// TIA Portal project "Bachelor _Project" (V17)
// By Soroush Tehranchi

(* hardware
DEVICE "S7-300/ET200M station_1"  S7-300 station
   slot 0: "Rail_0"  Rail  6ES7 390-1***0-0AA0
   slot 1: "PS 307 5A Outdoor_1"  PS 307 5A Outdoor  6ES7 307-1EA80-0AA0
   slot 1: "Rail_1"  Rail  6ES7 390-1***0-0AA0
   slot 1: "PS 307 5A_1"  PS 307 5A  6ES7 307-1EA01-0AA0
   slot 2: "PLC Siemens S7-300"  CPU 317-2 PN/DP  6ES7 317-2EK14-0AB0  V3.2
      slot 2: "PROFINET interface_1"  PN-IO
         slot 1: "Port_1"  Port
         slot 2: "Port_2"  Port
   slot 3: "IM 365_1"  IM 365  6ES7 365-0BA01-0AA0
      slot 1: "IM send/receive interface_1"  6ES7 365-0BA00-0AA0
   slot 3: "IM 365_1"  IM 365  6ES7 365-0BA01-0AA0
      slot 1: "IM send/receive interface_1"  6ES7 365-0BA00-0AA0
   slot 4: "DI 16x24VDC_1"  DI16 x 24VDC  6ES7 321-1BH02-0AA0
   slot 4: "DO 16x24VDC/0.5A_1"  DO16 x 24VDC / 0.5A  6ES7 322-1BH01-0AA0
   slot 5: "DI 16x24VDC_2"  DI16 x 24VDC  6ES7 321-1BH02-0AA0
   slot 5: "DO 16x24VDC/0.5A_2"  DO16 x 24VDC / 0.5A  6ES7 322-1BH01-0AA0
   slot 6: "DI 16x24VDC_3"  DI16 x 24VDC  6ES7 321-1BH02-0AA0
   slot 6: "DO 16x24VDC/0.5A_3"  DO16 x 24VDC / 0.5A  6ES7 322-1BH01-0AA0
   slot 7: "DI 16x24VDC_4"  DI16 x 24VDC  6ES7 321-1BH02-0AA0
   slot 7: "DO 16x24VDC/0.5A_4"  DO16 x 24VDC / 0.5A  6ES7 322-1BH01-0AA0
   slot 8: "AI 8x12BIT_1"  AI8 x 12 bits  6ES7 331-7KF02-0AB0
   slot 8: "FM 350-1 Counter_1"  FM 350-1 Counter  6ES7 350-1AH03-0AE0
   slot 9: "AI 8x12BIT_2"  AI8 x 12 bits  6ES7 331-7KF02-0AB0
   slot 9: "AI 8x12BIT_1"  AI8 x 12 bits  6ES7 331-7KF02-0AB0
   slot 10: "AI 8x12BIT_3"  AI8 x 12 bits  6ES7 331-7KF02-0AB0
   slot 10: "AI 8x12BIT_2"  AI8 x 12 bits  6ES7 331-7KF02-0AB0
   slot 11: "AO 8x12BIT_1"  AO8 x 12 bits  6ES7 332-5HF00-0AB0
   slot 11: "AO 8x12BIT_1"  AO8 x 12 bits  6ES7 332-5HF00-0AB0
DEVICE "HMI_1"  TP1200 Comfort
   slot 0: "HMI_1"  TP1200 Comfort  6AV2 124-0MC01-0AX0  17.0.0.0
   slot 1: "HMI_RT_1"  TP1200 Comfort  6AV2 124-0MC01-0AX0  17.0.0.0
   slot 5: "HMI_1.IE_CP_1"  PROFINET Interface  17.0.0.0
      slot 1: "PROFINET Interface_1"  PROFINET Interface
         slot 1: "Port_1"  Port
         slot 2: "Port_2"  Port
   slot 7: "HMI_1.MPI/DP_CP_1"  MPI/DP Interface  17.0.0.0
*)

// ===== PLC "PLC Siemens S7-300"  CPU 317-2 PN/DP =====

VAR_GLOBAL   // PLC tag table "Default tag table"
   "blue assembler convoyer timer" AT %T0 : Timer;
   "Machinings 2 timer(1)" AT %T1 : Timer;
   "Machinings 2 timer" AT %T2 : Timer;
   "Machinings 3 timer" AT %T3 : Timer;
   "Machinings 4 timer" AT %T4 : Timer;
   "station 1 counter" AT %C0 : Counter;
   "count sort line" AT %C1 : Counter;
   "count up sort" AT %M1.4 : Bool;
   "in position sort" AT %M1.5 : Bool;
   "Green base memory" AT %M1.6 : Bool;
   "sort convoyer edje" AT %M1.7 : Bool;
   "Green base counter" AT %C2 : Counter;
   "Blue base counter" AT %C3 : Counter;
   "Green lid counter" AT %C4 : Counter;
   "Blue lid counter" AT %C5 : Counter;
   "Green base counter number" AT %MW100 : Int;
   "Blue base counter number" AT %MW102 : Int;
   "Green lid counter number" AT %MW104 : Int;
   "Blue lid counter number" AT %MW106 : Int;
   "pusher edje 6" AT %M2.0 : Bool;
   "pusher edje 5" AT %M2.1 : Bool;
   "pusher edje 3" AT %M2.2 : Bool;
   "pusher edje 2" AT %M2.3 : Bool;
   "sort line counter number" AT %MW108 : Int;
   "encoder edje5" AT %M3.2 : Bool;
   "encoder edje6" AT %M3.3 : Bool;
   "encoder edje7" AT %M3.4 : Bool;
   "encoder edje8" AT %M3.5 : Bool;
   "encoder edje9" AT %M3.6 : Bool;
   "encoder edje10" AT %M3.7 : Bool;
   "encoder edje11" AT %M4.0 : Bool;
   "encoder edje12" AT %M4.1 : Bool;
   "encoder edje13" AT %M4.2 : Bool;
   "encoder edje14" AT %M4.3 : Bool;
   "encoder edje15" AT %M4.4 : Bool;
   "encoder edje16" AT %M4.5 : Bool;
   "Blue lid memory" AT %M4.6 : Bool;
   "green lid memory" AT %M4.7 : Bool;
   "initial assembler 2" AT %M6.7 : Bool;
   "initial assembler 1" AT %M6.6 : Bool;
   "Packaging Green  Clamp Sensor" AT %I3.6 : Bool;
   "green assembler convoyer timer" AT %T5 : Timer;
   "packing 1 uptimer" AT %T6 : Timer;
   "counter packing 1 uptime" AT %C6 : Counter;
   "Packing blue uptime" AT %T7 : Timer;
   "uptime blue packing" AT %C7 : Counter;
   "Item in blue pack" AT %C8 : Counter;
   "Item in green pack" AT %C9 : Counter;
   "Blue pack produced" AT %C10 : Counter;
   "green pack produced" AT %C11 : Counter;
   "blue product" AT %C12 : Counter;
   "green product" AT %C13 : Counter;
   "Assembler uptime blue" AT %T8 : Timer;
   "Blue Assembler uptime" AT %C14 : Counter;
   "green assembler uptimer" AT %T9 : Timer;
   "green assembler uptime" AT %C15 : Counter;
   "main convoyer uptimer" AT %T10 : Timer;
   "main convoyer uptime" AT %C16 : Counter;
   "crane uptimer" AT %T12 : Timer;
   "crane uptime" AT %C17 : Counter;
END_VAR

VAR_GLOBAL   // PLC tag table "Inputs"
   "Base  Blue Positioner (Clamped)" AT %I0.0 : Bool;
   "Base  Blue Positioner (Limit)" AT %I0.1 : Bool;
   "Base  Green Positioner (Clamped)" AT %I0.2 : Bool;
   "Base  Green Positioner (Limit)" AT %I0.3 : Bool;
   "Base Blue Clamp Sensor" AT %I0.4 : Bool;
   "Base Green Clamp Sensor" AT %I0.5 : Bool;
   "Blue Pusher Base  (Front Limit)" AT %I0.6 : Bool;
   "Blue Pusher Base (Back Limit)" AT %I0.7 : Bool;
   "Blue Pusher Lid (Back Limit)" AT %I1.0 : Bool;
   "Blue Pusher Lid (Front Limit)" AT %I1.1 : Bool;
   "Green Pusher Base  (Front Limit)" AT %I1.2 : Bool;
   "Green Pusher Base (Back Limit)" AT %I1.3 : Bool;
   "Green Pusher Lid (Back Limit)" AT %I1.4 : Bool;
   "Green Pusher Lid (Front Limit)" AT %I1.5 : Bool;
   "Lid  Blue Positioner (Clamped)" AT %I1.6 : Bool;
   "Lid  Green Positioner (Clamped)" AT %I1.7 : Bool;
   "Lid Blue Clamp Sensor" AT %I2.0 : Bool;
   "Lid Green Clamp Sensor" AT %I2.1 : Bool;
   "Machining Center 1 (Opened)" AT %I2.2 : Bool;
   "Machining Center 2 (Opened)" AT %I2.3 : Bool;
   "Machining Center 3 (Opened)" AT %I2.4 : Bool;
   "Machining Center 4 (Opened)" AT %I2.5 : Bool;
   "Machining Center 1 (Is Busy)" AT %I2.6 : Bool;
   "Machining Center 2 (Is Busy)" AT %I2.7 : Bool;
   "Machining Center 3 (Is Busy)" AT %I3.0 : Bool;
   "Machining Center 4 (Is Busy)" AT %I3.1 : Bool;
   "Packaging Blue (Limit)" AT %I3.2 : Bool;
   "Packaging Blue Palet Sensor" AT %I3.3 : Bool;
   "Packaging Blue(Clamped)" AT %I3.4 : Bool;
   "Packaging Green  (Limit)" AT %I3.5 : Bool;
   "Packaging Blue Clamp Sensor" AT %I3.7 : Bool;
   "Packaging Green  Palet Sensor" AT %I4.0 : Bool;
   "Packaging Green (Clamped)" AT %I4.1 : Bool;
   "Pick & Place 1 (C Limit) packaging" AT %I4.2 : Bool;
   "Pick & Place 2 (C Limit) packaging" AT %I4.3 : Bool;
   "Assmebler 1  grabed" AT %I4.4 : Bool;
   "Assmebler 2  grabed" AT %I4.5 : Bool;
   "Pick & Place 1 (Box Detected) packaging" AT %I5.4 : Bool;
   "Pick & Place 2 (Box Detected) packaging" AT %I5.5 : Bool;
   "Stacker Crane 1 Moving-X" AT %I6.2 : Bool;
   "Stacker Crane 1 Moving-Z" AT %I6.3 : Bool;
   "Stacker Crane 1 Left Limit" AT %I6.4 : Bool;
   "Stacker Crane 1 Right Limit" AT %I6.5 : Bool;
   "Stacker Crane 1 Middle Limit" AT %I6.6 : Bool;
   "Turntable 1 (Limit 0)" AT %I6.7 : Bool;
   "Turntable 1 (Limit 90)" AT %I7.0 : Bool;
   "Turntable 1 (Back Limit)" AT %I7.1 : Bool;
   "Turntable 1 (Front Limit)" AT %I7.2 : Bool;
   "Sort Convoyer Encoder Signal A" AT %I8.0 : Bool;
   "Sort Convoyer Encoder Signal B" AT %I8.1 : Bool;
   "Assemble Base Blue Convoyer" AT %Q0.1 : Bool;
   "Assemble Base Green Convoyer" AT %Q0.2 : Bool;
   "Assemble Lid Blue Convoyer" AT %Q0.3 : Bool;
   "Assemble Lid Green Convoyer" AT %Q0.4 : Bool;
   "Base  Blue Positioner  (Raise)" AT %Q0.5 : Bool;
   "Base  Blue Positioner (Clamp)" AT %Q0.6 : Bool;
   "Base  Green Positioner (Clamp)" AT %Q0.7 : Bool;
   "Base  Green Positioner (Raise)" AT %Q1.0 : Bool;
   "Blue Assemble Exit Convoyer 1" AT %Q1.1 : Bool;
   "Blue Assemble Exit Convoyer 2" AT %Q1.2 : Bool;
   "Blue Pusher Base" AT %Q1.3 : Bool;
   "Blue Pusher Lid" AT %Q1.4 : Bool;
   "Exit Convoyer" AT %Q1.5 : Bool;
   "Green Assemble Exit Convoyer" AT %Q1.6 : Bool;
   "Green Pusher Base" AT %Q1.7 : Bool;
   "Green Pusher Lid" AT %Q2.0 : Bool;
   "Lid  Blue Positioner (Clamp)" AT %Q2.2 : Bool;
   "Lid  Green Positioner (Clamp)" AT %Q2.3 : Bool;
   "Machining1 Exit Convoyer" AT %Q2.5 : Bool;
   "Machining2 Exit Convoyer" AT %Q2.6 : Bool;
   "Machining3 Exit Convoyer" AT %Q2.7 : Bool;
   "Machining4 Exit Convoyer" AT %Q3.0 : Bool;
   "Machining1 Entry Convoyer" AT %Q3.1 : Bool;
   "Machining2 Entry Convoyer" AT %Q3.2 : Bool;
   "Machining3 Entry Convoyer" AT %Q3.3 : Bool;
   "Machining4 Entry Convoyer" AT %Q3.4 : Bool;
   "Machinings Exit Convoyer 1" AT %Q3.5 : Bool;
   "Machinings Exit Convoyer 2" AT %Q3.6 : Bool;
   "Machinings Exit Convoyer 3" AT %Q3.7 : Bool;
   "Packaging Blue (Raise)" AT %Q4.0 : Bool;
   "Packaging Blue Convoyer" AT %Q4.1 : Bool;
   "Packaging Blue Exit Convoyer 1" AT %Q4.2 : Bool;
   "Packaging Blue Exit Convoyer 2" AT %Q4.3 : Bool;
   "Packaging Blue Exit Convoyer 3" AT %Q4.4 : Bool;
   "Packaging Blue(Clamp)" AT %Q4.5 : Bool;
   "Packaging Green (Clamp)" AT %Q4.6 : Bool;
   "Packaging Green (Raise)" AT %Q4.7 : Bool;
   "Packaging Green Convoyer" AT %Q5.0 : Bool;
   "Packaging Green Exit Convoyer" AT %Q5.1 : Bool;
   "Two-Axis Pick & Place 1 (Grab)" AT %Q5.2 : Bool;
   "Two-Axis Pick & Place 2 (Grab)" AT %Q5.3 : Bool;
   "Two-Axis Pick & Place 1 Rotate CW" AT %Q5.4 : Bool;
   "Pick & Place 1 C(+) packaging" AT %Q5.5 : Bool;
   "Pick & Place 2 C(+) packaging" AT %Q5.6 : Bool;
   "Pick & Place 1 (Grab) packaging" AT %Q5.7 : Bool;
   "Two-Axis Pick & Place 2 Rotate CW" AT %Q6.0 : Bool;
   "Two-Axis Pick & Place 1 Gripper CW" AT %Q6.1 : Bool;
   "Two-Axis Pick & Place 2 Gripper CW" AT %Q6.2 : Bool;
   "Pick & Place 2 (Grab) packaging" AT %Q6.6 : Bool;
   "Sort Convoyer" AT %Q6.7 : Bool;
   "Stacker Crane 1 Lift" AT %Q7.0 : Bool;
   "Stacker Crane 1 (Left)" AT %Q7.1 : Bool;
   "Stacker Crane 1 (Right)" AT %Q7.2 : Bool;
   "Turntable 1 Turn" AT %Q7.4 : Bool;
   "Turntable 1 Roll (+)" AT %Q7.5 : Bool;
   "Turntable 1 Roll (-)" AT %Q7.6 : Bool;
   "Vision Sensor 1 (Value)" AT %ID100 : DInt;
   "Pick & Place 2 Z Position (V) packaging" AT %ID104 : Real;
   "Pick & Place 2 Y Position (V) packaging" AT %ID108 : Real;
   "Pick & Place 2 X Position (V) packaging" AT %ID112 : Real;
   "Pick & Place 1 Z Position (V) packaging" AT %ID116 : Real;
   "Pick & Place 1 Y Position (V) packaging" AT %ID120 : Real;
   "Pick & Place 1 X Position (V) packaging" AT %ID124 : Real;
   "Machining Center 4 (Progress)" AT %ID128 : DInt;
   "Machining Center 3 (Progress)" AT %ID132 : DInt;
   "Machining Center 2 (Progress)" AT %ID136 : DInt;
   "Machining Center 1 (Progress)" AT %ID140 : DInt;
   "Vision Sensor 2 (Value)" AT %ID144 : DInt;
   "Vision Sensor 3 (Value)" AT %ID148 : DInt;
   "Vision Sensor 4 (Value)" AT %ID152 : DInt;
   "Two-Axis Pick & Place 1 X Position (V)" AT %ID156 : Real;
   "Two-Axis Pick & Place 1 Z Position (V)" AT %ID160 : Real;
   "Two-Axis Pick & Place 2 X Position (V)" AT %ID164 : Real;
   "Two-Axis Pick & Place 2 Z Position (V)" AT %ID168 : Real;
   "Pick & Place 1 Y Set Point(V) packaging" AT %QD100 : Real;
   "Pick & Place 2 Y Set Point(V) packaging" AT %QD104 : Real;
   "Pick & Place 1 X Set Point (V) packaging" AT %QD108 : Real;
   "Pick & Place 1 Z Set Point (V) packaging" AT %QD112 : Real;
   "Pick & Place 2 X Set Point (V) packaging" AT %QD116 : Real;
   "Pick & Place 2 Z Set Point (V) packaging" AT %QD120 : Real;
   "Stacker Crane 1 Target Position" AT %QD124 : DInt;
   "Two-Axis Pick & Place 1 X Set Point (V)" AT %QD128 : Real;
   "Two-Axis Pick & Place 1 Z Set Point (V)" AT %QD132 : Real;
   "Two-Axis Pick & Place 2 X Set Point (V)" AT %QD136 : Real;
   "Two-Axis Pick & Place 2 Z Set Point (V)" AT %QD140 : Real;
   "two axis  1 assembler rotating" AT %I4.6 : Bool;
   "two axis  2 assembler rotating" AT %I4.7 : Bool;
   "Capacitive Sensor Exit line 1" AT %I5.0 : Bool;
   "Capacitive Sensor Exit line 2" AT %I5.1 : Bool;
   "cran capacetive sensor" AT %I5.2 : Bool;
   "packaging to turn table convoyer" AT %Q2.1 : Bool;
   "Loading convoyer -" AT %Q0.0 : Bool;
   "Loading convoyer +" AT %Q2.4 : Bool;
   "Emitter 6" AT %Q6.3 : Bool;
   "Emmiter5" AT %Q6.4 : Bool;
END_VAR

VAR_GLOBAL   // PLC tag table "memory"
   "start_mach_entry_conv" AT %M0.0 : Bool;   // start machine center convoyer
   "reset convoyers" AT %M0.1 : Bool;
   "Machining Center busy1" AT %M0.2 : Bool;
   "Machining Center busy2" AT %M0.3 : Bool;
   "Machining Center busy3" AT %M0.4 : Bool;
   "Machining Center busy4" AT %M0.5 : Bool;
   "Machining Center busy1 convoyer" AT %M0.6 : Bool;
   "Machining Center busy2 convoyer" AT %M0.7 : Bool;
   "Machining Center busy3 convoyer" AT %M1.0 : Bool;
   "Machining Center busy4 convoyer" AT %M1.1 : Bool;
   "count down memory" AT %M1.2 : Bool;
   "count up memory" AT %M1.3 : Bool;
   "reset sorter" AT %M3.1 : Bool;
   "blue lid clamp sensor edje" AT %M5.0 : Bool;
   "blue base clamp sensor edje" AT %M5.1 : Bool;
   "green lid clamp sensor edje" AT %M5.2 : Bool;
   "green base clamp sensor edje" AT %M5.3 : Bool;
   "line 1 ready" AT %M5.4 : Bool;
   "line 2 ready" AT %M5.5 : Bool;
   "line 3 ready" AT %M5.6 : Bool;
   "line 4 ready" AT %M5.7 : Bool;
   "assemble 1 complet" AT %M6.0 : Bool;
   "assemble 2 complet" AT %M6.1 : Bool;
   "reset convoyers assembler" AT %M6.2 : Bool;
   "ready 1 edje" AT %M6.3 : Bool;
   "blue lid clamp sensor edje2" AT %M6.4 : Bool;
   "blue base positioner rise adje up" AT %M6.5 : Bool;
   "blue base positioner rise adje down" AT %M7.0 : Bool;
   "blue base clamp sensor edje2" AT %M7.1 : Bool;
   "green lid clamp sensor edje2" AT %M7.2 : Bool;
   "green  base positioner rise adje up" AT %M7.3 : Bool;
   "green base positioner rise adje down" AT %M7.4 : Bool;
   "green  base clamp sensor edje2" AT %M7.5 : Bool;
   "Packaging Green  Clamp Sensor edje" AT %M7.6 : Bool;
   "Packaging Green  Clamp Senso edje" AT %M7.7 : Bool;
   "packing 1 done" AT %M8.0 : Bool;
   "packing 2 done" AT %M8.1 : Bool;
   "Packaging Blue Palet Sensor edje" AT %M8.2 : Bool;
   "exit convoyer packing blue ready" AT %M8.3 : Bool;
   "entry convoyer packing blue ready" AT %M8.4 : Bool;
   "Packaging Blue Palet Sensor edje2" AT %M8.5 : Bool;
   "Packaging Green  Clamp Sensor edje 2" AT %M8.6 : Bool;
   "ready to pack 1" AT %M8.7 : Bool;
   "ready to pack 2" AT %M9.0 : Bool;
   "reset packer 1" AT %M9.1 : Bool;
   "reset packer 2" AT %M9.2 : Bool;
   "Capacitive Sensor Exit line 1 edje" AT %M9.3 : Bool;
   "Capacitive Sensor Exit line 2 edje" AT %M9.4 : Bool;
   "Packaging Blue Clamp Sensor edje 2" AT %M9.5 : Bool;
   "entry convoyer packing green ready" AT %M9.6 : Bool;
   "Packaging green Palet Sensor edje" AT %M9.7 : Bool;
   "exit convoyer packing green ready" AT %M10.0 : Bool;
   "Packaging green Palet Sensor edje2" AT %M10.1 : Bool;
   "Load to storage" AT %M10.2 : Bool;
   "Capacitive Sensor Exit line 2 edje(1)" AT %M10.3 : Bool;
   "deploy" AT %M10.4 : Bool;
   "user target position" AT %MD20 : DInt;
   "product type" AT %MW24 : Int;   // 0 empty 1green 2 blue
   "blue item stored" AT %MW26 : Int;
   "green item stored" AT %MW28 : Int;
   "cap" AT %MW30 : Int;
END_VAR

// folder: Packaging

DATA_BLOCK "Packaging system_DB"   // DB3
{ S7_Optimized_Access := 'FALSE' }
VERSION : 0.1
// stored: InstanceOfName Packaging systemBlue
"Packaging systemBlue"
BEGIN
END_DATA_BLOCK

DATA_BLOCK "Packaging system2_DB"   // DB4
{ S7_Optimized_Access := 'FALSE' }
VERSION : 0.1
// stored: InstanceOfName Packaging system Green
"Packaging system Green"
BEGIN
END_DATA_BLOCK

// folder: Sort And Assemble

DATA_BLOCK "Assembler_devic_DB"   // DB1
{ S7_Optimized_Access := 'FALSE' }
VERSION : 0.1
// stored: InstanceOfName Assembler_devic
"Assembler_devic"
BEGIN
END_DATA_BLOCK

DATA_BLOCK "Assembler_devic_DB_1"   // DB2
{ S7_Optimized_Access := 'FALSE' }
VERSION : 0.1
// stored: InstanceOfName Assembler_devic
"Assembler_devic"
BEGIN
END_DATA_BLOCK

// folder: Storage System

DATA_BLOCK "Turntable_DB"   // DB5
{ S7_Optimized_Access := 'FALSE' }
VERSION : 0.1
// stored: InstanceOfName Turntable
"Turntable"
BEGIN
END_DATA_BLOCK

DATA_BLOCK "Storage"   // DB6
{ S7_Optimized_Access := 'FALSE' }
VERSION : 0.1
   VAR
      status : Array[0..53] of Bool;
      cap : Int;
      "product type" : Array[0..53] of Int;
   END_VAR
BEGIN
   "product type"[1] := 0;
   "product type"[2] := 0;
END_DATA_BLOCK

DATA_BLOCK "stacker_DB"   // DB7
{ S7_Optimized_Access := 'FALSE' }
VERSION : 0.1
// stored: InstanceOfName stacker
"stacker"
BEGIN
END_DATA_BLOCK

// folder: (top level)

ORGANIZATION_BLOCK "Main"   // OB1, LAD
TITLE = "Main Program Sweep (Cycle)"
{ S7_Optimized_Access := 'FALSE' }
VERSION : 0.1
   VAR_TEMP
      OB1_EV_CLASS : Byte;   // Bits 0-3 = 1 (Coming event), Bits 4-7 = 1 (Event class 1)
      OB1_SCAN_1 : Byte;   // 1 (Cold restart scan 1 of OB 1), 3 (Scan 2-n of OB 1)
      OB1_PRIORITY : Byte;   // Priority of OB Execution
      OB1_OB_NUMBR : Byte;   // 1 (Organization block 1, OB1)
      OB1_RESERVED_1 : Byte;   // Reserved for system
      OB1_RESERVED_2 : Byte;   // Reserved for system
      OB1_PREV_CYCLE : Int;   // Cycle time of previous OB1 scan (milliseconds)
      OB1_MIN_CYCLE : Int;   // Minimum cycle time of OB1 (milliseconds)
      OB1_MAX_CYCLE : Int;   // Maximum cycle time of OB1 (milliseconds)
      OB1_DATE_TIME : Date_And_Time;   // Date and time OB1 started
   END_VAR
BEGIN

REGION Network 1: Machining Center
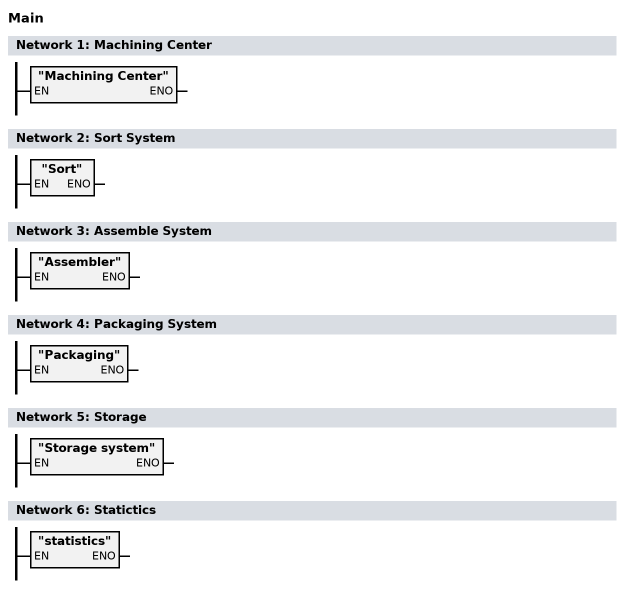
   RUNG wire#powerrail
      "Machining Center"()
   END_RUNG
   // the same network as SCL:
   "Machining Center"();
END_REGION

REGION Network 2: Sort System
   RUNG wire#powerrail
      "Sort"()
   END_RUNG
   // the same network as SCL:
   "Sort"();
END_REGION

REGION Network 3: Assemble System
   RUNG wire#powerrail
      "Assembler"()
   END_RUNG
   // the same network as SCL:
   "Assembler"();
END_REGION

REGION Network 4: Packaging System
   RUNG wire#powerrail
      "Packaging"()
   END_RUNG
   // the same network as SCL:
   "Packaging"();
END_REGION

REGION Network 5: Storage
   RUNG wire#powerrail
      "Storage system"()
   END_RUNG
   // the same network as SCL:
   "Storage system"();
END_REGION

REGION Network 6: Statictics
   RUNG wire#powerrail
      "statistics"()
   END_RUNG
   // the same network as SCL:
   "statistics"();
END_REGION
END_ORGANIZATION_BLOCK

// folder: Machining Center

FUNCTION "Machining Center" : Void   // FC1, LAD
TITLE = Machining Center
{ S7_Optimized_Access := 'FALSE' }
VERSION : 0.1
// This FC manage Entry Convoyer and exit convoyer
BEGIN

REGION Network 1: Entry Convoyers
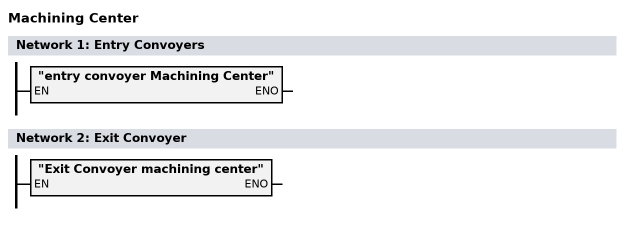
   RUNG wire#powerrail
      "entry convoyer Machining Center"()
   END_RUNG
   // the same network as SCL:
   "entry convoyer Machining Center"();
END_REGION

REGION Network 2: Exit Convoyer
   RUNG wire#powerrail
      "Exit Convoyer machining center"()
   END_RUNG
   // the same network as SCL:
   "Exit Convoyer machining center"();
END_REGION
END_FUNCTION

FUNCTION "entry convoyer Machining Center" : Void   // FC2, LAD
{ S7_Optimized_Access := 'FALSE' }
VERSION : 0.1
BEGIN

REGION Network 1
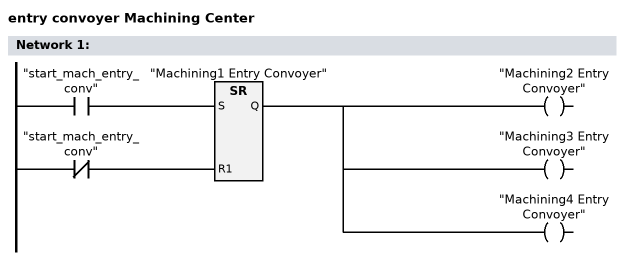
   RUNG wire#powerrail
      Contact( "start_mach_entry_conv" )
      S_SR(operand := "Machining1 Entry Convoyer", r1 := wire#w1)
      wire#w2
      Coil( "Machining2 Entry Convoyer" )
   END_RUNG
   RUNG wire#powerrail
      I_Contact( "start_mach_entry_conv" )
   END_RUNG wire#w1
   RUNG wire#w2
      Coil( "Machining3 Entry Convoyer" )
   END_RUNG
   RUNG wire#w2
      Coil( "Machining4 Entry Convoyer" )
   END_RUNG
   // the same network as SCL:
   IF "start_mach_entry_conv" THEN
       "Machining1 Entry Convoyer" := TRUE;   // SR flip-flop
   END_IF;
   IF NOT "start_mach_entry_conv" THEN "Machining1 Entry Convoyer" := FALSE; END_IF;
   "Machining2 Entry Convoyer" := "Machining1 Entry Convoyer";
   "Machining3 Entry Convoyer" := "Machining1 Entry Convoyer";
   "Machining4 Entry Convoyer" := "Machining1 Entry Convoyer";
END_REGION
END_FUNCTION

FUNCTION "Exit Convoyer machining center" : Void   // FC3, LAD
{ S7_Optimized_Access := 'FALSE' }
VERSION : 0.1
   VAR_TEMP   // added for the SCL form of the ladder/FBD networks
      _w1 : Bool;
      _w2 : Bool;
      _w3 : Bool;
      _w4 : Bool;
      _w5 : Bool;
      _w6 : Bool;
      _w7 : Bool;
      _w8 : Bool;
      _w9 : Bool;
      _w10 : Bool;
      _w11 : Bool;
      _s5time1 : S5Time;
   END_VAR
BEGIN

REGION Network 1: Exit Convoyers
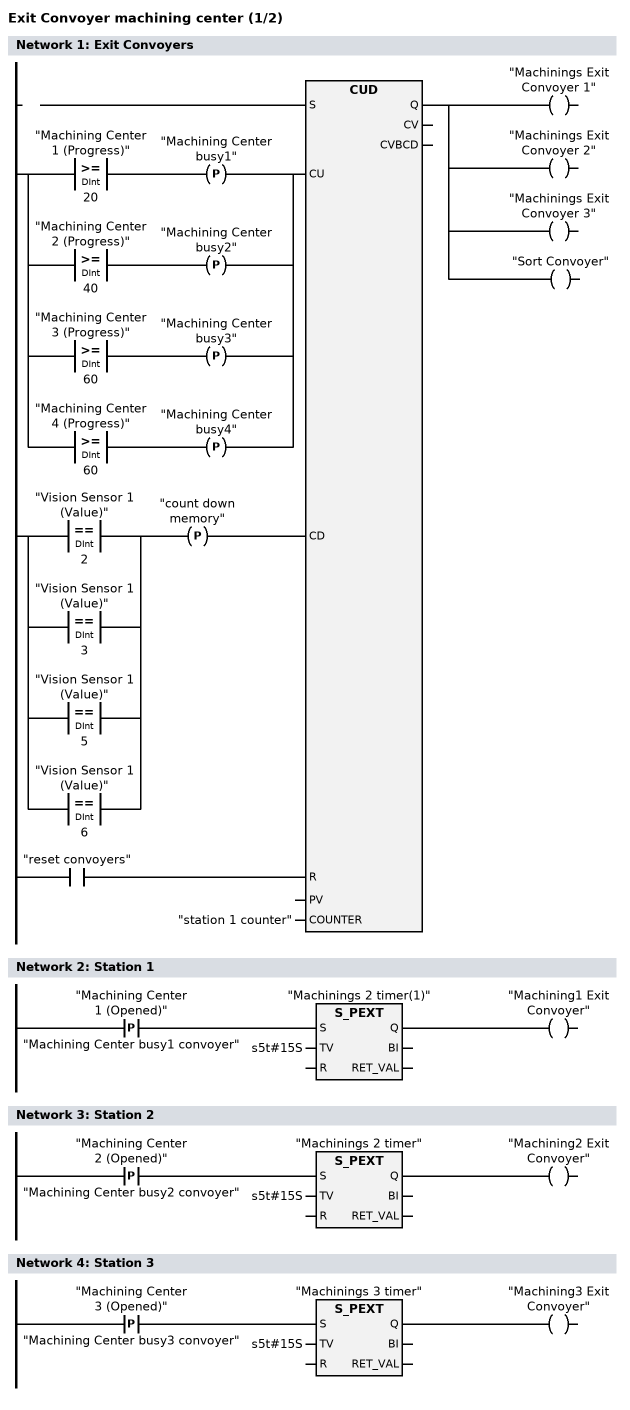
   // no SCL statement known for Cud: written as a call
   #_w1 := "Machining Center 1 (Progress)" >= 20;
   #_w2 := #_w1 AND NOT "Machining Center busy1";   // rising edge
   "Machining Center busy1" := #_w1;
   #_w3 := "Machining Center 2 (Progress)" >= 40;
   #_w4 := #_w3 AND NOT "Machining Center busy2";   // rising edge
   "Machining Center busy2" := #_w3;
   #_w5 := "Machining Center 3 (Progress)" >= 60;
   #_w6 := #_w5 AND NOT "Machining Center busy3";   // rising edge
   "Machining Center busy3" := #_w5;
   #_w7 := "Machining Center 4 (Progress)" >= 60;
   #_w8 := #_w7 AND NOT "Machining Center busy4";   // rising edge
   "Machining Center busy4" := #_w7;
   #_w9 := ("Vision Sensor 1 (Value)" = 2) OR ("Vision Sensor 1 (Value)" = 3) OR ("Vision Sensor 1 (Value)" = 5) OR ("Vision Sensor 1 (Value)" = 6);
   #_w10 := #_w9 AND NOT "count down memory";   // rising edge
   "count down memory" := #_w9;
   Cud(cu := #_w2 OR #_w4 OR #_w6 OR #_w8,
       cd := #_w10,
       r := "reset convoyers",
       "counter" := "station 1 counter",
       q => #_w11);
   "Machinings Exit Convoyer 1" := #_w11;
   "Machinings Exit Convoyer 2" := #_w11;
   "Machinings Exit Convoyer 3" := #_w11;
   "Sort Convoyer" := #_w11;
END_REGION

REGION Network 2: Station 1
   RUNG wire#powerrail
      P_Contact(operand := "Machining Center 1 (Opened)", bit := "Machining Center busy1 convoyer")
      S_PEXT(T_NO := "Machinings 2 timer(1)", TV := s5t#15S, R :=, BI =>, RET_VAL =>)
      Coil( "Machining1 Exit Convoyer" )
   END_RUNG
   // the same network as SCL:
   #_w1 := "Machining Center 1 (Opened)" AND NOT "Machining Center busy1 convoyer";   // rising edge of "Machining Center 1 (Opened)"
   "Machining Center busy1 convoyer" := "Machining Center 1 (Opened)";
   #_s5time1 := S_PEXT(T_NO := "Machinings 2 timer(1)", S := #_w1, TV := s5t#15S, Q => #_w2);
   "Machining1 Exit Convoyer" := #_w2;
END_REGION

REGION Network 3: Station 2
   RUNG wire#powerrail
      P_Contact(operand := "Machining Center 2 (Opened)", bit := "Machining Center busy2 convoyer")
      S_PEXT(T_NO := "Machinings 2 timer", TV := s5t#15S, R :=, BI =>, RET_VAL =>)
      Coil( "Machining2 Exit Convoyer" )
   END_RUNG
   // the same network as SCL:
   #_w1 := "Machining Center 2 (Opened)" AND NOT "Machining Center busy2 convoyer";   // rising edge of "Machining Center 2 (Opened)"
   "Machining Center busy2 convoyer" := "Machining Center 2 (Opened)";
   #_s5time1 := S_PEXT(T_NO := "Machinings 2 timer", S := #_w1, TV := s5t#15S, Q => #_w2);
   "Machining2 Exit Convoyer" := #_w2;
END_REGION

REGION Network 4: Station 3
   RUNG wire#powerrail
      P_Contact(operand := "Machining Center 3 (Opened)", bit := "Machining Center busy3 convoyer")
      S_PEXT(T_NO := "Machinings 3 timer", TV := s5t#15S, R :=, BI =>, RET_VAL =>)
      Coil( "Machining3 Exit Convoyer" )
   END_RUNG
   // the same network as SCL:
   #_w1 := "Machining Center 3 (Opened)" AND NOT "Machining Center busy3 convoyer";   // rising edge of "Machining Center 3 (Opened)"
   "Machining Center busy3 convoyer" := "Machining Center 3 (Opened)";
   #_s5time1 := S_PEXT(T_NO := "Machinings 3 timer", S := #_w1, TV := s5t#15S, Q => #_w2);
   "Machining3 Exit Convoyer" := #_w2;
END_REGION

REGION Network 5: Station 4
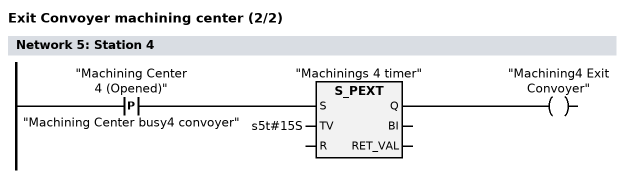
   RUNG wire#powerrail
      P_Contact(operand := "Machining Center 4 (Opened)", bit := "Machining Center busy4 convoyer")
      S_PEXT(T_NO := "Machinings 4 timer", TV := s5t#15S, R :=, BI =>, RET_VAL =>)
      Coil( "Machining4 Exit Convoyer" )
   END_RUNG
   // the same network as SCL:
   #_w1 := "Machining Center 4 (Opened)" AND NOT "Machining Center busy4 convoyer";   // rising edge of "Machining Center 4 (Opened)"
   "Machining Center busy4 convoyer" := "Machining Center 4 (Opened)";
   #_s5time1 := S_PEXT(T_NO := "Machinings 4 timer", S := #_w1, TV := s5t#15S, Q => #_w2);
   "Machining4 Exit Convoyer" := #_w2;
END_REGION
END_FUNCTION

// folder: Packaging

FUNCTION_BLOCK "Packaging systemBlue"   // FB2, GRAPH
{ S7_Optimized_Access := 'FALSE' }
VERSION : 0.1
   VAR_INPUT
      OFF_SQ : Bool := false;   // Turn sequence off
      INIT_SQ : Bool := false;   // Set sequence to initial state
      ACK_EF : Bool := false;   // Acknowledge all errors and faults
      S_PREV : Bool := false;   // Output previous step in parameter S_NO
      S_NEXT : Bool := false;   // Indicate next step in parameter S_NO
      SW_AUTO : Bool := false;   // Automatic mode
      SW_TAP : Bool := false;   // Semiautomatic/switch with transition
      SW_TOP : Bool := false;   // Semiautomatic/ignore transition
      SW_MAN : Bool := false;   // Manual mode
      S_SEL : Int := 0;   // Select step to be output to S_NO
      S_ON : Bool := false;   // Activate step indicated in S_NO
      S_OFF : Bool := false;   // Deactivate step indicated S_NO
      T_PUSH : Bool := false;   // Enable transition to switch in semi automatic mode
   END_VAR
   VAR_OUTPUT
      S_NO : Int := 0;   // Step number
      S_MORE : Bool := false;   // More steps are available and can be shown in S_NO
      S_ACTIVE : Bool := false;   // Step indicated in S_NO is active
      ERR_FLT : Bool := false;   // Interlock or supervision group error
      AUTO_ON : Bool := false;   // Automatic mode is active
      TAP_ON : Bool := false;   // Semiautomatic mode/step with transition enabled
      TOP_ON : Bool := false;   // Semiautomatic mode/ignore transition enabled
      MAN_ON : Bool := false;   // Manual mode is active
   END_VAR
   VAR_IN_OUT
      "packer x set point" : Real;
      "packer x value" : Real;
      "packer y set point" : Real;
      "packer y  value" : Real;
      "packer z set point" : Real;
      "packer z value" : Real;
      clamp : Bool;
      clamped : Bool;
      grab : Bool;
      grabed : Bool;
      "arm rotate" : Bool;
      ready : Bool;
      "convoyer entry ready" : Bool;
      "pack done" : Bool;
      "Exit convoyer" : Bool;
   END_VAR
   VAR
      SWITCH : Array[0..0] of DWord;
      SW_SQTS : Array[0..36] of Byte;
      SW_ADDR : Word := 16#24;
      G7T_0 : GraphTransition;
      G7S_0 : GraphStep;
      PRE_CRIT : Array[0..0] of DWord;
      POST_CRIT : Array[0..0] of DWord;
      TVX : Array[0..2] of Byte;
      TTX : Array[0..2] of Byte;
      TSX : Array[0..2] of Byte;
      S00X : Array[0..2] of Byte;
      SOFFX : Array[0..2] of Byte;
      SONX : Array[0..2] of Byte;
      SAX : Array[0..2] of Byte;
      SERRX : Array[0..37] of Byte;
      SMX : Array[0..37] of Byte;
      S0X : Array[0..37] of Byte;
      S1X : Array[0..37] of Byte;
      S_DISPLAY : Int;   // Internal display of output parameter S_NO
      S_SEL_OLD : Int;   // Previous value in S_SEL
      S_DISPIDX : Byte;   // Index of the step in S_NO
      T_DISPIDX : Byte;   // Index of the transition displayed in T_NO
      MOPEDGE : Struct
         AUTO : Bool := false;
         MAN : Bool := false;
         TAP : Bool := false;
         TOP : Bool := false;
         ACK_S : Bool := false;
         REG_S : Bool := false;
         T_PREV : Bool := false;
         T_NEXT : Bool := false;
         LOCK : Bool := false;
         SUP : Bool := false;
         ACKREQ : Bool := false;
         SSKIP : Bool := false;
         OFF : Bool := false;
         INIT : Bool := false;
         HALT : Bool := false;
         TMS_HALT : Bool := false;
         OPS_ZERO : Bool := false;
         SACT_DISP : Bool := false;
         SEF_DISP : Bool := false;
         SALL_DISP : Bool := false;
         S_PREV : Bool := false;
         S_NEXT : Bool := false;
         S_SELOK : Bool := false;
         S_ON : Bool := false;
         S_OFF : Bool := false;
         T_PUSH : Bool := false;
         REG : Bool := false;
         ACK : Bool := false;
         IL_PERM : Bool := false;
         T_PERM : Bool := false;
         ILP_MAN : Bool := false;
      END_STRUCT;
      MOP : Struct   // Mode
         AUTO : Bool := true;   // Status: automatic mode
         MAN : Bool := false;   // Status: manual mode
         TAP : Bool := false;   // Status: semi automatic/switch with transition
         TOP : Bool := false;   // Status: semi automatic/ignore transition
         ACK_S : Bool := false;   // Request: acknowledge step at parameter S_NO
         REG_S : Bool := false;   // Request: register step indicated in S_NO
         T_PREV : Bool := false;   // Request: output previous valid transition in T_NO
         T_NEXT : Bool := false;   // Request: output next valid transition in T_NO
         LOCK : Bool := true;   // Status: interlocks activated
         SUP : Bool := true;   // Status: supervisions activated
         ACKREQ : Bool := true;   // Status: acknowledgment required
         SSKIP : Bool := false;   // Status: "Skip steps" enabled
         OFF : Bool := false;   // Request: deactivate all steps
         INIT : Bool := true;   // Request: set sequence to initial state
         HALT : Bool := false;   // Status: sequence halted
         TMS_HALT : Bool := false;   // Status: all internal timers held
         OPS_ZERO : Bool := false;   // Status: set all operands processed with N, L, D instructions to 0
         SACT_DISP : Bool := true;   // Status: display active steps only
         SEF_DISP : Bool := false;   // Status: display only steps with errors and disrupted steps
         SALL_DISP : Bool := false;   // Status: display all steps
         S_PREV : Bool := false;   // Request: output previous step to S_NO
         S_NEXT : Bool := false;   // Request: Output next step at S_NO parameter
         S_SELOK : Bool := false;   // Request: output step number from S_SEL to S_NO
         S_ON : Bool := false;   // Request: activate step indicated in S_NO
         S_OFF : Bool := false;   // Request: deactivate step at parameter S_NO
         T_PUSH : Bool := false;   // Request: transition switching enabled
         REG : Bool := false;   // Request: register all interlock and supervision errors
         ACK : Bool := false;   // Request: acknowledge all interlock and supervision errors
         IL_PERM : Bool := false;   // Status: permanent processing of all interlocks
         T_PERM : Bool := false;   // Status: permanent processing of all transitions
         ILP_MAN : Bool := false;   // Status: permanent processing of all interlocks in manual mode
      END_STRUCT;
      TICKS : Struct   // Clock speeds
         DELTA : Time := T#0ms;   // Time difference between cycles
         OLD : Time := T#0ms;   // 10 ms clock counter value in last cycle
         NEW : Time := T#0ms;   // 10 ms clock counter value in this cycle
      END_STRUCT;
      SQ_FLAGS : Struct   // Sequence bit memory
         ERR_FLT : Bool := false;   // Interlock and supervision group error
         ERROR : Bool := false;   // Interlock group error
         FAULT : Bool := false;   // Supervision group error
         RT_FAIL : Bool := false;   // Runtime error
         NO_SNO : Bool := false;   // Requested step number not found
         NF_OFL : Bool := false;   // Overflow: too many ON or OFF requests
         SA_OFL : Bool := false;   // Overflow: too many steps active
         TV_OFL : Bool := false;   // Overflow: too many valid transitions
         MSG_OFL : Bool := false;   // Overflow: not enough system resources for ALARM_S
         NO_SWI : Bool := false;   // Do not switch in this cycle
         CYC_OP : Bool := false;   // Cyclic execution of the sequence after initialization
         AS_MSG : Bool := true;   // Alarms during runtime enabled or disabled by instruction
         AS_SEND : Bool := false;   // Send alarms from WR_USMSG or only enter in diagnostics buffer
         SQ_BUSY : Bool := false;   // Internal edge bit memory for sequence processing
         SA_BUSY : Bool := false;   // Internal edge bit memory for sequence processing
         AS_SIG : Bool := false;   // Edge bit memory for alarms from Alarm_S and Alarm_SQ
      END_STRUCT;
      S_PTR : DWord := 16#1500;
      S_PTR2 : DWord := 16#0;
      S_PTR3 : DWord := 16#3EB0;
      S_PTR4 : DWord := 16#3D80;
      T_PTR : DWord := 16#3C50;
      C_AR2 : DWord := 16#0;
      M_FBDB : DWord := 16#20000;
      M_SNO : Word := 16#0;
      M_EVID : Word := 16#0;
      M_EVIL : C_Alarm_s;
      M_EVSV : C_Alarm_s;
      M_EV : DWord := 16#3AC0;
      CRIT : Array[0..31] of Bool;
      S_START : Byte := 16#0;
      S_IDX : Byte := 16#0;
      S_INT : Int := 72;
      S_TMP : Byte := 16#0;
      T_START : Byte := 16#0;
      T_IDX : Byte := 16#0;
      T_TMP : Byte := 16#0;
      T_TMP2 : Byte := 16#00;
      TV_POT : Byte := 16#06;
      RETURN1 : Byte := 16#0;
      RETURN2 : Byte := 16#0;
      SINI : Array[0..2] of Byte;
      LSTT : Array[0..36] of Byte;
      ATAJ : Array[0..36] of Byte;
      ATAB : Array[0..36] of Byte;
      PSTT : Array[0..36] of Byte;
      NSTT : Array[0..36] of Byte;
      ASSJ : Array[0..36] of Byte;
      ASSB : Array[0..36] of Byte;
      PTTS : Array[0..36] of Byte;
      NTTS : Array[0..36] of Byte;
      PRE_CNT : Word := 16#1;
      POST_CNT : Word := 16#1;
      ADR_COND : Word := 16#0;
      MAX_TVAL : Byte := 16#1;
      MAX_SACT : Byte := 16#1;
      MAX_CRIT : Byte := 16#4;
      T_CNT : Byte := 16#24;
      SUP_CNT : Byte := 16#0;
      LOCK_CNT : Byte := 16#0;
      S_CNT : Byte := 16#24;
      SQ_CNT : Byte := 16#1;
      PRS_INPAR : DWord := 16#E000FEC8;
      PRS_OUTPAR : DWord := 16#E000800F;
      GC_FLAGS : Struct
         T_MACH : Byte := 16#EB;
         COND_ED : Byte := 16#E3;
         W_LEVEL : Byte := 16#D5;
         FB_IF : Byte := 16#FA;
         AS_MSG : Word := 16#404;
         SSB : Word := 16#108;
         DILG : Word := 16#9D6;
         ADDR_T0 : Word := 16#50;
         CRIT_AVAIL : Bool := false;
         SSKIP_AVAIL : Bool := true;
         SSKIP_ON : Bool := false;
         ACK_REQ : Bool := true;
         SYNC_AVAIL : Bool := true;
         ILP_MAN : Bool := false;
         SWM_LOCKED : Bool := false;
         SAVE_SW : Bool := true;
      END_STRUCT;
      G7_FBMARK : Byte := 16#3C;
      G7_RELEASE : Byte := 16#3C;
      G7_ID2 : Byte := 16#37;
      G7_ID1 : Byte := 16#47;
   END_VAR
   // SW_SQTS[0] := 16#1;
   // TVX[0] := 16#1;
   // TTX[0] := 16#1;
   // TSX[0] := 16#1;
   // S00X[0] := 16#1;
   // SOFFX[0] := 16#1;
   // SONX[0] := 16#1;
   // SAX[0] := 16#1;
   // SERRX[0] := 16#1;
   // SMX[0] := 16#1;
   // S0X[0] := 16#1;
   // S1X[0] := 16#1;
   // SINI[0] := 16#2;
   // SINI[1] := 16#1;
   // SINI[2] := 0;
   // LSTT[0] := 0;
   // LSTT[1] := 0;
   // LSTT[2] := 0;
   // LSTT[3] := 0;
   // LSTT[4] := 0;
   // LSTT[5] := 0;
   // LSTT[6] := 0;
   // LSTT[7] := 0;
   // LSTT[8] := 0;
   // LSTT[9] := 0;
   // LSTT[10] := 0;
   // LSTT[11] := 0;
   // LSTT[12] := 0;
   // LSTT[13] := 0;
   // LSTT[14] := 0;
   // LSTT[15] := 0;
   // LSTT[16] := 0;
   // LSTT[17] := 0;
   // LSTT[18] := 0;
   // LSTT[19] := 0;
   // LSTT[20] := 0;
   // LSTT[21] := 0;
   // LSTT[22] := 0;
   // LSTT[23] := 0;
   // LSTT[24] := 0;
   // LSTT[25] := 0;
   // LSTT[26] := 0;
   // LSTT[27] := 0;
   // LSTT[28] := 0;
   // LSTT[29] := 0;
   // LSTT[30] := 0;
   // LSTT[31] := 0;
   // LSTT[32] := 16#1;
   // ATAJ[0] := 0;
   // ATAJ[1] := 16#1;
   // ATAJ[2] := 16#2;
   // ATAJ[3] := 16#3;
   // ATAJ[4] := 16#4;
   // ATAJ[5] := 16#5;
   // ATAJ[6] := 16#6;
   // ATAJ[7] := 16#7;
   // ATAJ[8] := 16#8;
   // ATAJ[9] := 16#9;
   // ATAJ[10] := 16#A;
   // ATAJ[11] := 16#B;
   // ATAJ[12] := 16#C;
   // ATAJ[13] := 16#D;
   // ATAJ[14] := 16#E;
   // ATAJ[15] := 16#F;
   // ATAJ[16] := 16#10;
   // ATAJ[17] := 16#11;
   // ATAJ[18] := 16#12;
   // ATAJ[19] := 16#13;
   // ATAJ[20] := 16#14;
   // ATAJ[21] := 16#15;
   // ATAJ[22] := 16#16;
   // ATAJ[23] := 16#17;
   // ATAJ[24] := 16#18;
   // ATAJ[25] := 16#19;
   // ATAJ[26] := 16#1A;
   // ATAJ[27] := 16#1B;
   // ATAJ[28] := 16#1C;
   // ATAJ[29] := 16#1D;
   // ATAJ[30] := 16#1E;
   // ATAJ[31] := 16#1F;
   // ATAJ[32] := 16#20;
   // ATAB[0] := 0;
   // ATAB[1] := 16#1;
   // ATAB[2] := 16#2;
   // ATAB[3] := 16#3;
   // ATAB[4] := 16#4;
   // ATAB[5] := 16#5;
   // ATAB[6] := 16#6;
   // ATAB[7] := 16#7;
   // ATAB[8] := 16#8;
   // ATAB[9] := 16#9;
   // ATAB[10] := 16#A;
   // ATAB[11] := 16#B;
   // ATAB[12] := 16#C;
   // ATAB[13] := 16#D;
   // ATAB[14] := 16#E;
   // ATAB[15] := 16#F;
   // ATAB[16] := 16#10;
   // ATAB[17] := 16#11;
   // ATAB[18] := 16#12;
   // ATAB[19] := 16#13;
   // ATAB[20] := 16#14;
   // ATAB[21] := 16#15;
   // ATAB[22] := 16#16;
   // ATAB[23] := 16#17;
   // ATAB[24] := 16#18;
   // ATAB[25] := 16#19;
   // ATAB[26] := 16#1A;
   // ATAB[27] := 16#1B;
   // ATAB[28] := 16#1C;
   // ATAB[29] := 16#1D;
   // ATAB[30] := 16#1E;
   // ATAB[31] := 16#1F;
   // ATAB[32] := 16#20;
   // PSTT[0] := 0;
   // PSTT[1] := 16#1;
   // PSTT[2] := 16#2;
   // PSTT[3] := 16#3;
   // PSTT[4] := 16#4;
   // PSTT[5] := 16#5;
   // PSTT[6] := 16#6;
   // PSTT[7] := 16#7;
   // PSTT[8] := 16#8;
   // PSTT[9] := 16#9;
   // PSTT[10] := 16#A;
   // PSTT[11] := 16#B;
   // PSTT[12] := 16#C;
   // PSTT[13] := 16#D;
   // PSTT[14] := 16#E;
   // PSTT[15] := 16#F;
   // PSTT[16] := 16#10;
   // PSTT[17] := 16#11;
   // PSTT[18] := 16#12;
   // PSTT[19] := 16#13;
   // PSTT[20] := 16#14;
   // PSTT[21] := 16#15;
   // PSTT[22] := 16#16;
   // PSTT[23] := 16#17;
   // PSTT[24] := 16#18;
   // PSTT[25] := 16#19;
   // PSTT[26] := 16#1A;
   // PSTT[27] := 16#1B;
   // PSTT[28] := 16#1C;
   // PSTT[29] := 16#1D;
   // PSTT[30] := 16#1E;
   // PSTT[31] := 16#1F;
   // PSTT[32] := 16#20;
   // NSTT[0] := 16#1;
   // NSTT[1] := 16#2;
   // NSTT[2] := 16#3;
   // NSTT[3] := 16#4;
   // NSTT[4] := 16#5;
   // NSTT[5] := 16#6;
   // NSTT[6] := 16#21;
   // NSTT[7] := 16#8;
   // NSTT[8] := 16#9;
   // NSTT[9] := 16#A;
   // NSTT[10] := 16#B;
   // NSTT[11] := 16#C;
   // NSTT[12] := 16#D;
   // NSTT[13] := 16#E;
   // NSTT[14] := 16#22;
   // NSTT[15] := 16#10;
   // NSTT[16] := 16#11;
   // NSTT[17] := 16#12;
   // NSTT[18] := 16#13;
   // NSTT[19] := 16#14;
   // NSTT[20] := 16#15;
   // NSTT[21] := 16#16;
   // NSTT[22] := 16#23;
   // NSTT[23] := 16#18;
   // NSTT[24] := 16#19;
   // NSTT[25] := 16#1A;
   // NSTT[26] := 16#1B;
   // NSTT[27] := 16#1C;
   // NSTT[28] := 16#1D;
   // NSTT[29] := 16#1E;
   // NSTT[30] := 16#24;
   // NSTT[31] := 16#20;
   // NSTT[32] := 16#1;
   // ASSJ[0] := 0;
   // ASSJ[1] := 16#1;
   // ASSJ[2] := 16#2;
   // ASSJ[3] := 16#3;
   // ASSJ[4] := 16#4;
   // ASSJ[5] := 16#5;
   // ASSJ[6] := 16#6;
   // ASSJ[7] := 16#7;
   // ASSJ[8] := 16#8;
   // ASSJ[9] := 16#9;
   // ASSJ[10] := 16#A;
   // ASSJ[11] := 16#B;
   // ASSJ[12] := 16#C;
   // ASSJ[13] := 16#D;
   // ASSJ[14] := 16#E;
   // ASSJ[15] := 16#F;
   // ASSJ[16] := 16#10;
   // ASSJ[17] := 16#11;
   // ASSJ[18] := 16#12;
   // ASSJ[19] := 16#13;
   // ASSJ[20] := 16#14;
   // ASSJ[21] := 16#15;
   // ASSJ[22] := 16#16;
   // ASSJ[23] := 16#17;
   // ASSJ[24] := 16#18;
   // ASSJ[25] := 16#19;
   // ASSJ[26] := 16#1A;
   // ASSJ[27] := 16#1B;
   // ASSJ[28] := 16#1C;
   // ASSJ[29] := 16#1D;
   // ASSJ[30] := 16#1E;
   // ASSJ[31] := 16#1F;
   // ASSJ[32] := 16#20;
   // ASSB[0] := 0;
   // ASSB[1] := 16#1;
   // ASSB[2] := 16#2;
   // ASSB[3] := 16#3;
   // ASSB[4] := 16#4;
   // ASSB[5] := 16#5;
   // ASSB[6] := 16#6;
   // ASSB[7] := 16#7;
   // ASSB[8] := 16#8;
   // ASSB[9] := 16#9;
   // ASSB[10] := 16#A;
   // ASSB[11] := 16#B;
   // ASSB[12] := 16#C;
   // ASSB[13] := 16#D;
   // ASSB[14] := 16#E;
   // ASSB[15] := 16#F;
   // ASSB[16] := 16#10;
   // ASSB[17] := 16#11;
   // ASSB[18] := 16#12;
   // ASSB[19] := 16#13;
   // ASSB[20] := 16#14;
   // ASSB[21] := 16#15;
   // ASSB[22] := 16#16;
   // ASSB[23] := 16#17;
   // ASSB[24] := 16#18;
   // ASSB[25] := 16#19;
   // ASSB[26] := 16#1A;
   // ASSB[27] := 16#1B;
   // ASSB[28] := 16#1C;
   // ASSB[29] := 16#1D;
   // ASSB[30] := 16#1E;
   // ASSB[31] := 16#1F;
   // ASSB[32] := 16#20;
   // PTTS[0] := 0;
   // PTTS[2] := 16#1;
   // PTTS[3] := 16#2;
   // PTTS[4] := 16#3;
   // PTTS[5] := 16#4;
   // PTTS[6] := 16#5;
   // PTTS[7] := 16#21;
   // PTTS[8] := 16#7;
   // PTTS[9] := 16#8;
   // PTTS[10] := 16#9;
   // PTTS[11] := 16#A;
   // PTTS[12] := 16#B;
   // PTTS[13] := 16#C;
   // PTTS[14] := 16#D;
   // PTTS[15] := 16#22;
   // PTTS[16] := 16#F;
   // PTTS[17] := 16#10;
   // PTTS[18] := 16#11;
   // PTTS[19] := 16#12;
   // PTTS[20] := 16#13;
   // PTTS[21] := 16#14;
   // PTTS[22] := 16#15;
   // PTTS[23] := 16#23;
   // PTTS[24] := 16#17;
   // PTTS[25] := 16#18;
   // PTTS[26] := 16#19;
   // PTTS[27] := 16#1A;
   // PTTS[28] := 16#1B;
   // PTTS[29] := 16#1C;
   // PTTS[30] := 16#1D;
   // PTTS[31] := 16#24;
   // PTTS[32] := 16#1F;
   // NTTS[0] := 0;
   // NTTS[1] := 16#1;
   // NTTS[2] := 16#2;
   // NTTS[3] := 16#3;
   // NTTS[4] := 16#4;
   // NTTS[5] := 16#5;
   // NTTS[6] := 16#6;
   // NTTS[7] := 16#7;
   // NTTS[8] := 16#8;
   // NTTS[9] := 16#9;
   // NTTS[10] := 16#A;
   // NTTS[11] := 16#B;
   // NTTS[12] := 16#C;
   // NTTS[13] := 16#D;
   // NTTS[14] := 16#E;
   // NTTS[15] := 16#F;
   // NTTS[16] := 16#10;
   // NTTS[17] := 16#11;
   // NTTS[18] := 16#12;
   // NTTS[19] := 16#13;
   // NTTS[20] := 16#14;
   // NTTS[21] := 16#15;
   // NTTS[22] := 16#16;
   // NTTS[23] := 16#17;
   // NTTS[24] := 16#18;
   // NTTS[25] := 16#19;
   // NTTS[26] := 16#1A;
   // NTTS[27] := 16#1B;
   // NTTS[28] := 16#1C;
   // NTTS[29] := 16#1D;
   // NTTS[30] := 16#1E;
   // NTTS[31] := 16#1F;
   // NTTS[32] := 16#20;
   // LSTT[33] := 0;
   // LSTT[34] := 0;
   // LSTT[35] := 0;
   // LSTT[36] := 0;
   // ATAJ[33] := 16#21;
   // ATAJ[34] := 16#22;
   // ATAJ[35] := 16#23;
   // ATAJ[36] := 16#24;
   // ATAB[33] := 16#21;
   // ATAB[34] := 16#22;
   // ATAB[35] := 16#23;
   // ATAB[36] := 16#24;
   // PSTT[33] := 16#21;
   // PSTT[34] := 16#22;
   // PSTT[35] := 16#23;
   // PSTT[36] := 16#24;
   // NSTT[33] := 16#7;
   // NSTT[34] := 16#F;
   // NSTT[35] := 16#17;
   // NSTT[36] := 16#1F;
   // ASSJ[33] := 16#21;
   // ASSJ[34] := 16#22;
   // ASSJ[35] := 16#23;
   // ASSJ[36] := 16#24;
   // ASSB[33] := 16#21;
   // ASSB[34] := 16#22;
   // ASSB[35] := 16#23;
   // ASSB[36] := 16#24;
   // PTTS[33] := 16#6;
   // PTTS[34] := 16#E;
   // PTTS[35] := 16#16;
   // PTTS[36] := 16#1E;
   // NTTS[33] := 16#21;
   // NTTS[34] := 16#22;
   // NTTS[35] := 16#23;
   // NTTS[36] := 16#24;
BEGIN
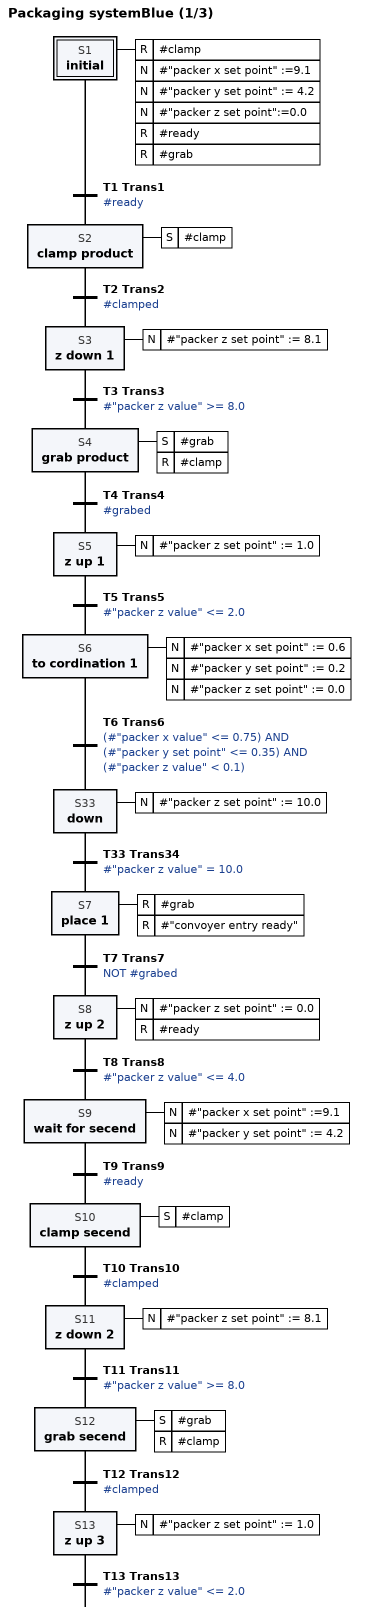
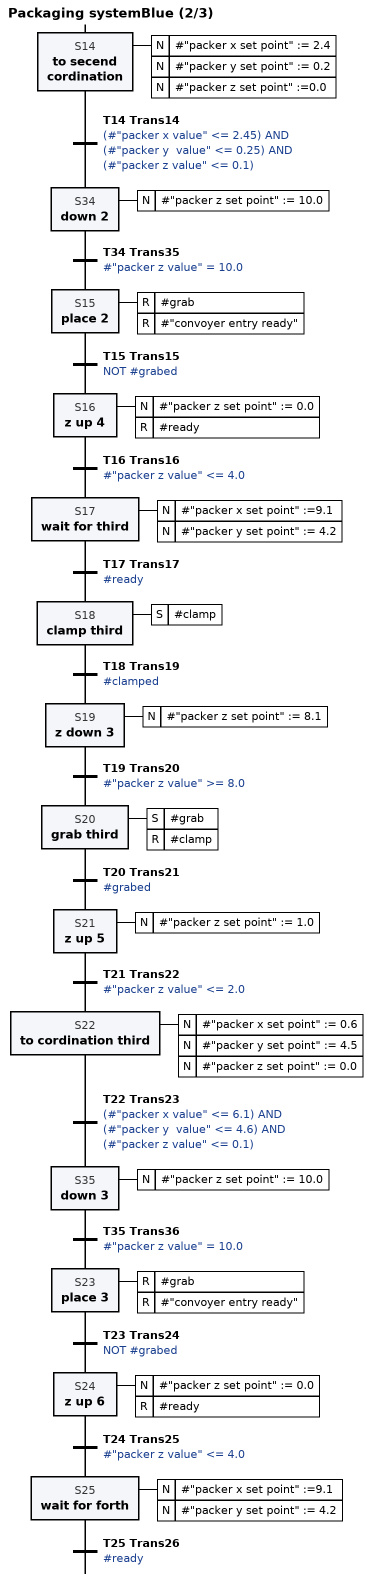
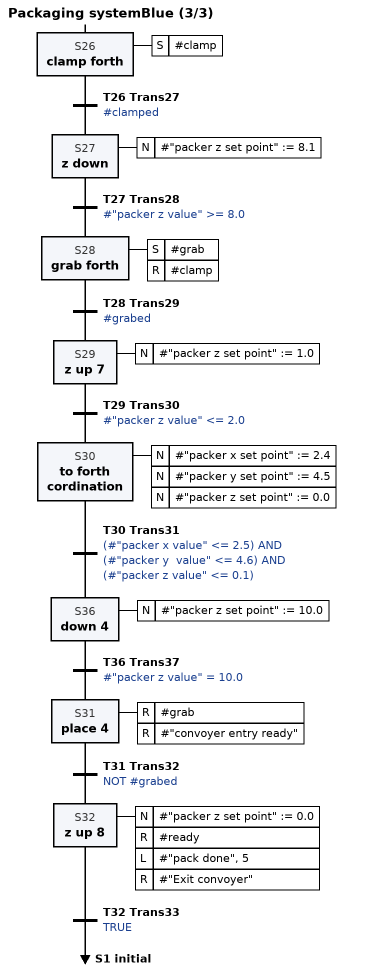
   // sequencer 1
   INITIAL_STEP initial:   // S1
              R    #clamp
              N    #"packer x set point" :=9.1
              N    #"packer y set point" := 4.2
              N    #"packer z set point":=0.0
              R    #ready
              R    #grab
   END_STEP
   TRANSITION Trans1 FROM initial TO "clamp product"   // T1
      := #ready;
   END_TRANSITION
   STEP "clamp product":   // S2
              S    #clamp
   END_STEP
   TRANSITION Trans2 FROM "clamp product" TO "z down 1"   // T2
      := #clamped;
   END_TRANSITION
   STEP "z down 1":   // S3
              N    #"packer z set point" := 8.1
   END_STEP
   TRANSITION Trans3 FROM "z down 1" TO "grab product"   // T3
      := #"packer z value" >= 8.0;
   END_TRANSITION
   STEP "grab product":   // S4
              S    #grab
              R    #clamp
   END_STEP
   TRANSITION Trans4 FROM "grab product" TO "z up 1"   // T4
      := #grabed;
   END_TRANSITION
   STEP "z up 1":   // S5
              N    #"packer z set point" := 1.0
   END_STEP
   TRANSITION Trans5 FROM "z up 1" TO "to cordination 1"   // T5
      := #"packer z value" <= 2.0;
   END_TRANSITION
   STEP "to cordination 1":   // S6
              N    #"packer x set point" := 0.6
              N    #"packer y set point" := 0.2
              N    #"packer z set point" := 0.0
   END_STEP
   TRANSITION Trans6 FROM "to cordination 1" TO down   // T6
      := (#"packer x value" <= 0.75) AND (#"packer y set point" <= 0.35) AND (#"packer z value" < 0.1);
   END_TRANSITION
   STEP "place 1":   // S7
              R    #grab
              R    #"convoyer entry ready"
   END_STEP
   TRANSITION Trans7 FROM "place 1" TO "z up 2"   // T7
      := NOT #grabed;
   END_TRANSITION
   STEP "z up 2":   // S8
              N    #"packer z set point" := 0.0
              R    #ready
   END_STEP
   TRANSITION Trans8 FROM "z up 2" TO "wait for secend"   // T8
      := #"packer z value" <= 4.0;
   END_TRANSITION
   STEP "wait for secend":   // S9
              N    #"packer x set point" :=9.1
              N    #"packer y set point" := 4.2
   END_STEP
   TRANSITION Trans9 FROM "wait for secend" TO "clamp secend"   // T9
      := #ready;
   END_TRANSITION
   STEP "clamp secend":   // S10
              S    #clamp
   END_STEP
   TRANSITION Trans10 FROM "clamp secend" TO "z down 2"   // T10
      := #clamped;
   END_TRANSITION
   STEP "z down 2":   // S11
              N    #"packer z set point" := 8.1
   END_STEP
   TRANSITION Trans11 FROM "z down 2" TO "grab secend"   // T11
      := #"packer z value" >= 8.0;
   END_TRANSITION
   STEP "grab secend":   // S12
              S    #grab
              R    #clamp
   END_STEP
   TRANSITION Trans12 FROM "grab secend" TO "z up 3"   // T12
      := #clamped;
   END_TRANSITION
   STEP "z up 3":   // S13
              N    #"packer z set point" := 1.0
   END_STEP
   TRANSITION Trans13 FROM "z up 3" TO "to secend cordination"   // T13
      := #"packer z value" <= 2.0;
   END_TRANSITION
   STEP "to secend cordination":   // S14
              N    #"packer x set point" := 2.4
              N    #"packer y set point" := 0.2
              N    #"packer z set point" :=0.0
   END_STEP
   TRANSITION Trans14 FROM "to secend cordination" TO "down 2"   // T14
      := (#"packer x value" <= 2.45) AND (#"packer y  value" <= 0.25) AND (#"packer z value" <= 0.1);
   END_TRANSITION
   STEP "place 2":   // S15
              R    #grab
              R    #"convoyer entry ready"
   END_STEP
   TRANSITION Trans15 FROM "place 2" TO "z up 4"   // T15
      := NOT #grabed;
   END_TRANSITION
   STEP "z up 4":   // S16
              N    #"packer z set point" := 0.0
              R    #ready
   END_STEP
   TRANSITION Trans16 FROM "z up 4" TO "wait for third"   // T16
      := #"packer z value" <= 4.0;
   END_TRANSITION
   STEP "wait for third":   // S17
              N    #"packer x set point" :=9.1
              N    #"packer y set point" := 4.2
   END_STEP
   TRANSITION Trans17 FROM "wait for third" TO "clamp third"   // T17
      := #ready;
   END_TRANSITION
   STEP "grab third":   // S20
              S    #grab
              R    #clamp
   END_STEP
   TRANSITION Trans21 FROM "grab third" TO "z up 5"   // T20
      := #grabed;
   END_TRANSITION
   STEP "clamp third":   // S18
              S    #clamp
   END_STEP
   TRANSITION Trans19 FROM "clamp third" TO "z down 3"   // T18
      := #clamped;
   END_TRANSITION
   STEP "z down 3":   // S19
              N    #"packer z set point" := 8.1
   END_STEP
   TRANSITION Trans20 FROM "z down 3" TO "grab third"   // T19
      := #"packer z value" >= 8.0;
   END_TRANSITION
   STEP "z up 5":   // S21
              N    #"packer z set point" := 1.0
   END_STEP
   TRANSITION Trans22 FROM "z up 5" TO "to cordination third"   // T21
      := #"packer z value" <= 2.0;
   END_TRANSITION
   STEP "to cordination third":   // S22
              N    #"packer x set point" := 0.6
              N    #"packer y set point" := 4.5
              N    #"packer z set point" := 0.0
   END_STEP
   TRANSITION Trans23 FROM "to cordination third" TO "down 3"   // T22
      := (#"packer x value" <= 6.1) AND (#"packer y  value" <= 4.6) AND (#"packer z value" <= 0.1);
   END_TRANSITION
   STEP "place 3":   // S23
              R    #grab
              R    #"convoyer entry ready"
   END_STEP
   TRANSITION Trans24 FROM "place 3" TO "z up 6"   // T23
      := NOT #grabed;
   END_TRANSITION
   STEP "z up 6":   // S24
              N    #"packer z set point" := 0.0
              R    #ready
   END_STEP
   TRANSITION Trans25 FROM "z up 6" TO "wait for forth"   // T24
      := #"packer z value" <= 4.0;
   END_TRANSITION
   STEP "wait for forth":   // S25
              N    #"packer x set point" :=9.1
              N    #"packer y set point" := 4.2
   END_STEP
   TRANSITION Trans26 FROM "wait for forth" TO "clamp forth"   // T25
      := #ready;
   END_TRANSITION
   STEP "clamp forth":   // S26
              S    #clamp
   END_STEP
   TRANSITION Trans27 FROM "clamp forth" TO "z down"   // T26
      := #clamped;
   END_TRANSITION
   STEP "z down":   // S27
              N    #"packer z set point" := 8.1
   END_STEP
   TRANSITION Trans28 FROM "z down" TO "grab forth"   // T27
      := #"packer z value" >= 8.0;
   END_TRANSITION
   STEP "grab forth":   // S28
              S    #grab
              R    #clamp
   END_STEP
   TRANSITION Trans29 FROM "grab forth" TO "z up 7"   // T28
      := #grabed;
   END_TRANSITION
   STEP "z up 7":   // S29
              N    #"packer z set point" := 1.0
   END_STEP
   TRANSITION Trans30 FROM "z up 7" TO "to forth cordination"   // T29
      := #"packer z value" <= 2.0;
   END_TRANSITION
   STEP "to forth cordination":   // S30
              N    #"packer x set point" := 2.4
              N    #"packer y set point" := 4.5
              N    #"packer z set point" := 0.0
   END_STEP
   TRANSITION Trans31 FROM "to forth cordination" TO "down 4"   // T30
      := (#"packer x value" <= 2.5) AND (#"packer y  value" <= 4.6) AND (#"packer z value" <= 0.1);
   END_TRANSITION
   STEP "place 4":   // S31
              R    #grab
              R    #"convoyer entry ready"
   END_STEP
   TRANSITION Trans32 FROM "place 4" TO "z up 8"   // T31
      := NOT #grabed;
   END_TRANSITION
   STEP "z up 8":   // S32
              N    #"packer z set point" := 0.0
              R    #ready
              L    #"pack done", 5
              R    #"Exit convoyer"
   END_STEP
   TRANSITION Trans33 FROM "z up 8" TO initial   // T32, jump
      := TRUE;
   END_TRANSITION
   STEP down:   // S33
              N    #"packer z set point" := 10.0
   END_STEP
   TRANSITION Trans34 FROM down TO "place 1"   // T33
      := #"packer z value" = 10.0;
   END_TRANSITION
   STEP "down 2":   // S34
              N    #"packer z set point" := 10.0
   END_STEP
   TRANSITION Trans35 FROM "down 2" TO "place 2"   // T34
      := #"packer z value" = 10.0;
   END_TRANSITION
   STEP "down 3":   // S35
              N    #"packer z set point" := 10.0
   END_STEP
   TRANSITION Trans36 FROM "down 3" TO "place 3"   // T35
      := #"packer z value" = 10.0;
   END_TRANSITION
   STEP "down 4":   // S36
              N    #"packer z set point" := 10.0
   END_STEP
   TRANSITION Trans37 FROM "down 4" TO "place 4"   // T36
      := #"packer z value" = 10.0;
   END_TRANSITION
END_FUNCTION_BLOCK

FUNCTION_BLOCK "Packaging system Green"   // FB3, GRAPH
{ S7_Optimized_Access := 'FALSE' }
VERSION : 0.1
   VAR_INPUT
      OFF_SQ : Bool := false;   // Turn sequence off
      INIT_SQ : Bool := false;   // Set sequence to initial state
      ACK_EF : Bool := false;   // Acknowledge all errors and faults
      S_PREV : Bool := false;   // Output previous step in parameter S_NO
      S_NEXT : Bool := false;   // Indicate next step in parameter S_NO
      SW_AUTO : Bool := false;   // Automatic mode
      SW_TAP : Bool := false;   // Semiautomatic/switch with transition
      SW_TOP : Bool := false;   // Semiautomatic/ignore transition
      SW_MAN : Bool := false;   // Manual mode
      S_SEL : Int := 0;   // Select step to be output to S_NO
      S_ON : Bool := false;   // Activate step indicated in S_NO
      S_OFF : Bool := false;   // Deactivate step indicated S_NO
      T_PUSH : Bool := false;   // Enable transition to switch in semi automatic mode
   END_VAR
   VAR_OUTPUT
      S_NO : Int := 0;   // Step number
      S_MORE : Bool := false;   // More steps are available and can be shown in S_NO
      S_ACTIVE : Bool := false;   // Step indicated in S_NO is active
      ERR_FLT : Bool := false;   // Interlock or supervision group error
      AUTO_ON : Bool := false;   // Automatic mode is active
      TAP_ON : Bool := false;   // Semiautomatic mode/step with transition enabled
      TOP_ON : Bool := false;   // Semiautomatic mode/ignore transition enabled
      MAN_ON : Bool := false;   // Manual mode is active
   END_VAR
   VAR_IN_OUT
      "packer x set point" : Real;
      "packer x value" : Real;
      "packer y set point" : Real;
      "packer y  value" : Real;
      "packer z set point" : Real;
      "packer z value" : Real;
      clamp : Bool;
      clamped : Bool;
      grab : Bool;
      grabed : Bool;
      "arm rotate" : Bool;
      ready : Bool;
      "convoyer entry ready" : Bool;
      "pack done" : Bool;
      "Exit convoyer" : Bool;
   END_VAR
   VAR
      SWITCH : Array[0..0] of DWord;
      SW_SQTS : Array[0..36] of Byte;
      SW_ADDR : Word := 16#24;
      G7T_0 : GraphTransition;
      G7S_0 : GraphStep;
      PRE_CRIT : Array[0..0] of DWord;
      POST_CRIT : Array[0..0] of DWord;
      TVX : Array[0..2] of Byte;
      TTX : Array[0..2] of Byte;
      TSX : Array[0..2] of Byte;
      S00X : Array[0..2] of Byte;
      SOFFX : Array[0..2] of Byte;
      SONX : Array[0..2] of Byte;
      SAX : Array[0..2] of Byte;
      SERRX : Array[0..37] of Byte;
      SMX : Array[0..37] of Byte;
      S0X : Array[0..37] of Byte;
      S1X : Array[0..37] of Byte;
      S_DISPLAY : Int;   // Internal display of output parameter S_NO
      S_SEL_OLD : Int;   // Previous value in S_SEL
      S_DISPIDX : Byte;   // Index of the step in S_NO
      T_DISPIDX : Byte;   // Index of the transition displayed in T_NO
      MOPEDGE : Struct
         AUTO : Bool := false;
         MAN : Bool := false;
         TAP : Bool := false;
         TOP : Bool := false;
         ACK_S : Bool := false;
         REG_S : Bool := false;
         T_PREV : Bool := false;
         T_NEXT : Bool := false;
         LOCK : Bool := false;
         SUP : Bool := false;
         ACKREQ : Bool := false;
         SSKIP : Bool := false;
         OFF : Bool := false;
         INIT : Bool := false;
         HALT : Bool := false;
         TMS_HALT : Bool := false;
         OPS_ZERO : Bool := false;
         SACT_DISP : Bool := false;
         SEF_DISP : Bool := false;
         SALL_DISP : Bool := false;
         S_PREV : Bool := false;
         S_NEXT : Bool := false;
         S_SELOK : Bool := false;
         S_ON : Bool := false;
         S_OFF : Bool := false;
         T_PUSH : Bool := false;
         REG : Bool := false;
         ACK : Bool := false;
         IL_PERM : Bool := false;
         T_PERM : Bool := false;
         ILP_MAN : Bool := false;
      END_STRUCT;
      MOP : Struct   // Mode
         AUTO : Bool := true;   // Status: automatic mode
         MAN : Bool := false;   // Status: manual mode
         TAP : Bool := false;   // Status: semi automatic/switch with transition
         TOP : Bool := false;   // Status: semi automatic/ignore transition
         ACK_S : Bool := false;   // Request: acknowledge step at parameter S_NO
         REG_S : Bool := false;   // Request: register step indicated in S_NO
         T_PREV : Bool := false;   // Request: output previous valid transition in T_NO
         T_NEXT : Bool := false;   // Request: output next valid transition in T_NO
         LOCK : Bool := true;   // Status: interlocks activated
         SUP : Bool := true;   // Status: supervisions activated
         ACKREQ : Bool := true;   // Status: acknowledgment required
         SSKIP : Bool := false;   // Status: "Skip steps" enabled
         OFF : Bool := false;   // Request: deactivate all steps
         INIT : Bool := true;   // Request: set sequence to initial state
         HALT : Bool := false;   // Status: sequence halted
         TMS_HALT : Bool := false;   // Status: all internal timers held
         OPS_ZERO : Bool := false;   // Status: set all operands processed with N, L, D instructions to 0
         SACT_DISP : Bool := true;   // Status: display active steps only
         SEF_DISP : Bool := false;   // Status: display only steps with errors and disrupted steps
         SALL_DISP : Bool := false;   // Status: display all steps
         S_PREV : Bool := false;   // Request: output previous step to S_NO
         S_NEXT : Bool := false;   // Request: Output next step at S_NO parameter
         S_SELOK : Bool := false;   // Request: output step number from S_SEL to S_NO
         S_ON : Bool := false;   // Request: activate step indicated in S_NO
         S_OFF : Bool := false;   // Request: deactivate step at parameter S_NO
         T_PUSH : Bool := false;   // Request: transition switching enabled
         REG : Bool := false;   // Request: register all interlock and supervision errors
         ACK : Bool := false;   // Request: acknowledge all interlock and supervision errors
         IL_PERM : Bool := false;   // Status: permanent processing of all interlocks
         T_PERM : Bool := false;   // Status: permanent processing of all transitions
         ILP_MAN : Bool := false;   // Status: permanent processing of all interlocks in manual mode
      END_STRUCT;
      TICKS : Struct   // Clock speeds
         DELTA : Time := T#0ms;   // Time difference between cycles
         OLD : Time := T#0ms;   // 10 ms clock counter value in last cycle
         NEW : Time := T#0ms;   // 10 ms clock counter value in this cycle
      END_STRUCT;
      SQ_FLAGS : Struct   // Sequence bit memory
         ERR_FLT : Bool := false;   // Interlock and supervision group error
         ERROR : Bool := false;   // Interlock group error
         FAULT : Bool := false;   // Supervision group error
         RT_FAIL : Bool := false;   // Runtime error
         NO_SNO : Bool := false;   // Requested step number not found
         NF_OFL : Bool := false;   // Overflow: too many ON or OFF requests
         SA_OFL : Bool := false;   // Overflow: too many steps active
         TV_OFL : Bool := false;   // Overflow: too many valid transitions
         MSG_OFL : Bool := false;   // Overflow: not enough system resources for ALARM_S
         NO_SWI : Bool := false;   // Do not switch in this cycle
         CYC_OP : Bool := false;   // Cyclic execution of the sequence after initialization
         AS_MSG : Bool := true;   // Alarms during runtime enabled or disabled by instruction
         AS_SEND : Bool := false;   // Send alarms from WR_USMSG or only enter in diagnostics buffer
         SQ_BUSY : Bool := false;   // Internal edge bit memory for sequence processing
         SA_BUSY : Bool := false;   // Internal edge bit memory for sequence processing
         AS_SIG : Bool := false;   // Edge bit memory for alarms from Alarm_S and Alarm_SQ
      END_STRUCT;
      S_PTR : DWord := 16#1500;
      S_PTR2 : DWord := 16#0;
      S_PTR3 : DWord := 16#3EB0;
      S_PTR4 : DWord := 16#3D80;
      T_PTR : DWord := 16#3C50;
      C_AR2 : DWord := 16#0;
      M_FBDB : DWord := 16#30000;
      M_SNO : Word := 16#0;
      M_EVID : Word := 16#0;
      M_EVIL : C_Alarm_s;
      M_EVSV : C_Alarm_s;
      M_EV : DWord := 16#3AC0;
      CRIT : Array[0..31] of Bool;
      S_START : Byte := 16#0;
      S_IDX : Byte := 16#0;
      S_INT : Int := 72;
      S_TMP : Byte := 16#0;
      T_START : Byte := 16#0;
      T_IDX : Byte := 16#0;
      T_TMP : Byte := 16#0;
      T_TMP2 : Byte := 16#00;
      TV_POT : Byte := 16#06;
      RETURN1 : Byte := 16#0;
      RETURN2 : Byte := 16#0;
      SINI : Array[0..2] of Byte;
      LSTT : Array[0..36] of Byte;
      ATAJ : Array[0..36] of Byte;
      ATAB : Array[0..36] of Byte;
      PSTT : Array[0..36] of Byte;
      NSTT : Array[0..36] of Byte;
      ASSJ : Array[0..36] of Byte;
      ASSB : Array[0..36] of Byte;
      PTTS : Array[0..36] of Byte;
      NTTS : Array[0..36] of Byte;
      PRE_CNT : Word := 16#1;
      POST_CNT : Word := 16#1;
      ADR_COND : Word := 16#0;
      MAX_TVAL : Byte := 16#1;
      MAX_SACT : Byte := 16#1;
      MAX_CRIT : Byte := 16#4;
      T_CNT : Byte := 16#24;
      SUP_CNT : Byte := 16#0;
      LOCK_CNT : Byte := 16#0;
      S_CNT : Byte := 16#24;
      SQ_CNT : Byte := 16#1;
      PRS_INPAR : DWord := 16#E000FEC8;
      PRS_OUTPAR : DWord := 16#E000800F;
      GC_FLAGS : Struct
         T_MACH : Byte := 16#EB;
         COND_ED : Byte := 16#E3;
         W_LEVEL : Byte := 16#D5;
         FB_IF : Byte := 16#FA;
         AS_MSG : Word := 16#404;
         SSB : Word := 16#108;
         DILG : Word := 16#9D6;
         ADDR_T0 : Word := 16#50;
         CRIT_AVAIL : Bool := false;
         SSKIP_AVAIL : Bool := true;
         SSKIP_ON : Bool := false;
         ACK_REQ : Bool := true;
         SYNC_AVAIL : Bool := true;
         ILP_MAN : Bool := false;
         SWM_LOCKED : Bool := false;
         SAVE_SW : Bool := true;
      END_STRUCT;
      G7_FBMARK : Byte := 16#3C;
      G7_RELEASE : Byte := 16#3C;
      G7_ID2 : Byte := 16#37;
      G7_ID1 : Byte := 16#47;
   END_VAR
   // SW_SQTS[0] := 16#1;
   // TVX[0] := 16#1;
   // TTX[0] := 16#1;
   // TSX[0] := 16#1;
   // S00X[0] := 16#1;
   // SOFFX[0] := 16#1;
   // SONX[0] := 16#1;
   // SAX[0] := 16#1;
   // SERRX[0] := 16#1;
   // SMX[0] := 16#1;
   // S0X[0] := 16#1;
   // S1X[0] := 16#1;
   // SINI[0] := 16#2;
   // SINI[1] := 16#1;
   // SINI[2] := 0;
   // LSTT[0] := 0;
   // LSTT[1] := 0;
   // LSTT[2] := 0;
   // LSTT[3] := 0;
   // LSTT[4] := 0;
   // LSTT[5] := 0;
   // LSTT[6] := 0;
   // LSTT[7] := 0;
   // LSTT[8] := 0;
   // LSTT[9] := 0;
   // LSTT[10] := 0;
   // LSTT[11] := 0;
   // LSTT[12] := 0;
   // LSTT[13] := 0;
   // LSTT[14] := 0;
   // LSTT[15] := 0;
   // LSTT[16] := 0;
   // LSTT[17] := 0;
   // LSTT[18] := 0;
   // LSTT[19] := 0;
   // LSTT[20] := 0;
   // LSTT[21] := 0;
   // LSTT[22] := 0;
   // LSTT[23] := 0;
   // LSTT[24] := 0;
   // LSTT[25] := 0;
   // LSTT[26] := 0;
   // LSTT[27] := 0;
   // LSTT[28] := 0;
   // LSTT[29] := 0;
   // LSTT[30] := 0;
   // LSTT[31] := 0;
   // LSTT[32] := 16#1;
   // ATAJ[0] := 0;
   // ATAJ[1] := 16#1;
   // ATAJ[2] := 16#2;
   // ATAJ[3] := 16#3;
   // ATAJ[4] := 16#4;
   // ATAJ[5] := 16#5;
   // ATAJ[6] := 16#6;
   // ATAJ[7] := 16#7;
   // ATAJ[8] := 16#8;
   // ATAJ[9] := 16#9;
   // ATAJ[10] := 16#A;
   // ATAJ[11] := 16#B;
   // ATAJ[12] := 16#C;
   // ATAJ[13] := 16#D;
   // ATAJ[14] := 16#E;
   // ATAJ[15] := 16#F;
   // ATAJ[16] := 16#10;
   // ATAJ[17] := 16#11;
   // ATAJ[18] := 16#12;
   // ATAJ[19] := 16#13;
   // ATAJ[20] := 16#14;
   // ATAJ[21] := 16#15;
   // ATAJ[22] := 16#16;
   // ATAJ[23] := 16#17;
   // ATAJ[24] := 16#18;
   // ATAJ[25] := 16#19;
   // ATAJ[26] := 16#1A;
   // ATAJ[27] := 16#1B;
   // ATAJ[28] := 16#1C;
   // ATAJ[29] := 16#1D;
   // ATAJ[30] := 16#1E;
   // ATAJ[31] := 16#1F;
   // ATAJ[32] := 16#20;
   // ATAB[0] := 0;
   // ATAB[1] := 16#1;
   // ATAB[2] := 16#2;
   // ATAB[3] := 16#3;
   // ATAB[4] := 16#4;
   // ATAB[5] := 16#5;
   // ATAB[6] := 16#6;
   // ATAB[7] := 16#7;
   // ATAB[8] := 16#8;
   // ATAB[9] := 16#9;
   // ATAB[10] := 16#A;
   // ATAB[11] := 16#B;
   // ATAB[12] := 16#C;
   // ATAB[13] := 16#D;
   // ATAB[14] := 16#E;
   // ATAB[15] := 16#F;
   // ATAB[16] := 16#10;
   // ATAB[17] := 16#11;
   // ATAB[18] := 16#12;
   // ATAB[19] := 16#13;
   // ATAB[20] := 16#14;
   // ATAB[21] := 16#15;
   // ATAB[22] := 16#16;
   // ATAB[23] := 16#17;
   // ATAB[24] := 16#18;
   // ATAB[25] := 16#19;
   // ATAB[26] := 16#1A;
   // ATAB[27] := 16#1B;
   // ATAB[28] := 16#1C;
   // ATAB[29] := 16#1D;
   // ATAB[30] := 16#1E;
   // ATAB[31] := 16#1F;
   // ATAB[32] := 16#20;
   // PSTT[0] := 0;
   // PSTT[1] := 16#1;
   // PSTT[2] := 16#2;
   // PSTT[3] := 16#3;
   // PSTT[4] := 16#4;
   // PSTT[5] := 16#5;
   // PSTT[6] := 16#6;
   // PSTT[7] := 16#7;
   // PSTT[8] := 16#8;
   // PSTT[9] := 16#9;
   // PSTT[10] := 16#A;
   // PSTT[11] := 16#B;
   // PSTT[12] := 16#C;
   // PSTT[13] := 16#D;
   // PSTT[14] := 16#E;
   // PSTT[15] := 16#F;
   // PSTT[16] := 16#10;
   // PSTT[17] := 16#11;
   // PSTT[18] := 16#12;
   // PSTT[19] := 16#13;
   // PSTT[20] := 16#14;
   // PSTT[21] := 16#15;
   // PSTT[22] := 16#16;
   // PSTT[23] := 16#17;
   // PSTT[24] := 16#18;
   // PSTT[25] := 16#19;
   // PSTT[26] := 16#1A;
   // PSTT[27] := 16#1B;
   // PSTT[28] := 16#1C;
   // PSTT[29] := 16#1D;
   // PSTT[30] := 16#1E;
   // PSTT[31] := 16#1F;
   // PSTT[32] := 16#20;
   // NSTT[0] := 16#1;
   // NSTT[1] := 16#2;
   // NSTT[2] := 16#3;
   // NSTT[3] := 16#4;
   // NSTT[4] := 16#5;
   // NSTT[5] := 16#6;
   // NSTT[6] := 16#21;
   // NSTT[7] := 16#8;
   // NSTT[8] := 16#9;
   // NSTT[9] := 16#A;
   // NSTT[10] := 16#B;
   // NSTT[11] := 16#C;
   // NSTT[12] := 16#D;
   // NSTT[13] := 16#E;
   // NSTT[14] := 16#22;
   // NSTT[15] := 16#10;
   // NSTT[16] := 16#11;
   // NSTT[17] := 16#12;
   // NSTT[18] := 16#13;
   // NSTT[19] := 16#14;
   // NSTT[20] := 16#15;
   // NSTT[21] := 16#16;
   // NSTT[22] := 16#23;
   // NSTT[23] := 16#18;
   // NSTT[24] := 16#19;
   // NSTT[25] := 16#1A;
   // NSTT[26] := 16#1B;
   // NSTT[27] := 16#1C;
   // NSTT[28] := 16#1D;
   // NSTT[29] := 16#1E;
   // NSTT[30] := 16#24;
   // NSTT[31] := 16#20;
   // NSTT[32] := 16#1;
   // ASSJ[0] := 0;
   // ASSJ[1] := 16#1;
   // ASSJ[2] := 16#2;
   // ASSJ[3] := 16#3;
   // ASSJ[4] := 16#4;
   // ASSJ[5] := 16#5;
   // ASSJ[6] := 16#6;
   // ASSJ[7] := 16#7;
   // ASSJ[8] := 16#8;
   // ASSJ[9] := 16#9;
   // ASSJ[10] := 16#A;
   // ASSJ[11] := 16#B;
   // ASSJ[12] := 16#C;
   // ASSJ[13] := 16#D;
   // ASSJ[14] := 16#E;
   // ASSJ[15] := 16#F;
   // ASSJ[16] := 16#10;
   // ASSJ[17] := 16#11;
   // ASSJ[18] := 16#12;
   // ASSJ[19] := 16#13;
   // ASSJ[20] := 16#14;
   // ASSJ[21] := 16#15;
   // ASSJ[22] := 16#16;
   // ASSJ[23] := 16#17;
   // ASSJ[24] := 16#18;
   // ASSJ[25] := 16#19;
   // ASSJ[26] := 16#1A;
   // ASSJ[27] := 16#1B;
   // ASSJ[28] := 16#1C;
   // ASSJ[29] := 16#1D;
   // ASSJ[30] := 16#1E;
   // ASSJ[31] := 16#1F;
   // ASSJ[32] := 16#20;
   // ASSB[0] := 0;
   // ASSB[1] := 16#1;
   // ASSB[2] := 16#2;
   // ASSB[3] := 16#3;
   // ASSB[4] := 16#4;
   // ASSB[5] := 16#5;
   // ASSB[6] := 16#6;
   // ASSB[7] := 16#7;
   // ASSB[8] := 16#8;
   // ASSB[9] := 16#9;
   // ASSB[10] := 16#A;
   // ASSB[11] := 16#B;
   // ASSB[12] := 16#C;
   // ASSB[13] := 16#D;
   // ASSB[14] := 16#E;
   // ASSB[15] := 16#F;
   // ASSB[16] := 16#10;
   // ASSB[17] := 16#11;
   // ASSB[18] := 16#12;
   // ASSB[19] := 16#13;
   // ASSB[20] := 16#14;
   // ASSB[21] := 16#15;
   // ASSB[22] := 16#16;
   // ASSB[23] := 16#17;
   // ASSB[24] := 16#18;
   // ASSB[25] := 16#19;
   // ASSB[26] := 16#1A;
   // ASSB[27] := 16#1B;
   // ASSB[28] := 16#1C;
   // ASSB[29] := 16#1D;
   // ASSB[30] := 16#1E;
   // ASSB[31] := 16#1F;
   // ASSB[32] := 16#20;
   // PTTS[0] := 0;
   // PTTS[2] := 16#1;
   // PTTS[3] := 16#2;
   // PTTS[4] := 16#3;
   // PTTS[5] := 16#4;
   // PTTS[6] := 16#5;
   // PTTS[7] := 16#21;
   // PTTS[8] := 16#7;
   // PTTS[9] := 16#8;
   // PTTS[10] := 16#9;
   // PTTS[11] := 16#A;
   // PTTS[12] := 16#B;
   // PTTS[13] := 16#C;
   // PTTS[14] := 16#D;
   // PTTS[15] := 16#22;
   // PTTS[16] := 16#F;
   // PTTS[17] := 16#10;
   // PTTS[18] := 16#11;
   // PTTS[19] := 16#12;
   // PTTS[20] := 16#13;
   // PTTS[21] := 16#14;
   // PTTS[22] := 16#15;
   // PTTS[23] := 16#23;
   // PTTS[24] := 16#17;
   // PTTS[25] := 16#18;
   // PTTS[26] := 16#19;
   // PTTS[27] := 16#1A;
   // PTTS[28] := 16#1B;
   // PTTS[29] := 16#1C;
   // PTTS[30] := 16#1D;
   // PTTS[31] := 16#24;
   // PTTS[32] := 16#1F;
   // NTTS[0] := 0;
   // NTTS[1] := 16#1;
   // NTTS[2] := 16#2;
   // NTTS[3] := 16#3;
   // NTTS[4] := 16#4;
   // NTTS[5] := 16#5;
   // NTTS[6] := 16#6;
   // NTTS[7] := 16#7;
   // NTTS[8] := 16#8;
   // NTTS[9] := 16#9;
   // NTTS[10] := 16#A;
   // NTTS[11] := 16#B;
   // NTTS[12] := 16#C;
   // NTTS[13] := 16#D;
   // NTTS[14] := 16#E;
   // NTTS[15] := 16#F;
   // NTTS[16] := 16#10;
   // NTTS[17] := 16#11;
   // NTTS[18] := 16#12;
   // NTTS[19] := 16#13;
   // NTTS[20] := 16#14;
   // NTTS[21] := 16#15;
   // NTTS[22] := 16#16;
   // NTTS[23] := 16#17;
   // NTTS[24] := 16#18;
   // NTTS[25] := 16#19;
   // NTTS[26] := 16#1A;
   // NTTS[27] := 16#1B;
   // NTTS[28] := 16#1C;
   // NTTS[29] := 16#1D;
   // NTTS[30] := 16#1E;
   // NTTS[31] := 16#1F;
   // NTTS[32] := 16#20;
   // LSTT[33] := 0;
   // LSTT[34] := 0;
   // LSTT[35] := 0;
   // LSTT[36] := 0;
   // ATAJ[33] := 16#21;
   // ATAJ[34] := 16#22;
   // ATAJ[35] := 16#23;
   // ATAJ[36] := 16#24;
   // ATAB[33] := 16#21;
   // ATAB[34] := 16#22;
   // ATAB[35] := 16#23;
   // ATAB[36] := 16#24;
   // PSTT[33] := 16#21;
   // PSTT[34] := 16#22;
   // PSTT[35] := 16#23;
   // PSTT[36] := 16#24;
   // NSTT[33] := 16#7;
   // NSTT[34] := 16#F;
   // NSTT[35] := 16#17;
   // NSTT[36] := 16#1F;
   // ASSJ[33] := 16#21;
   // ASSJ[34] := 16#22;
   // ASSJ[35] := 16#23;
   // ASSJ[36] := 16#24;
   // ASSB[33] := 16#21;
   // ASSB[34] := 16#22;
   // ASSB[35] := 16#23;
   // ASSB[36] := 16#24;
   // PTTS[33] := 16#6;
   // PTTS[34] := 16#E;
   // PTTS[35] := 16#16;
   // PTTS[36] := 16#1E;
   // NTTS[33] := 16#21;
   // NTTS[34] := 16#22;
   // NTTS[35] := 16#23;
   // NTTS[36] := 16#24;
BEGIN
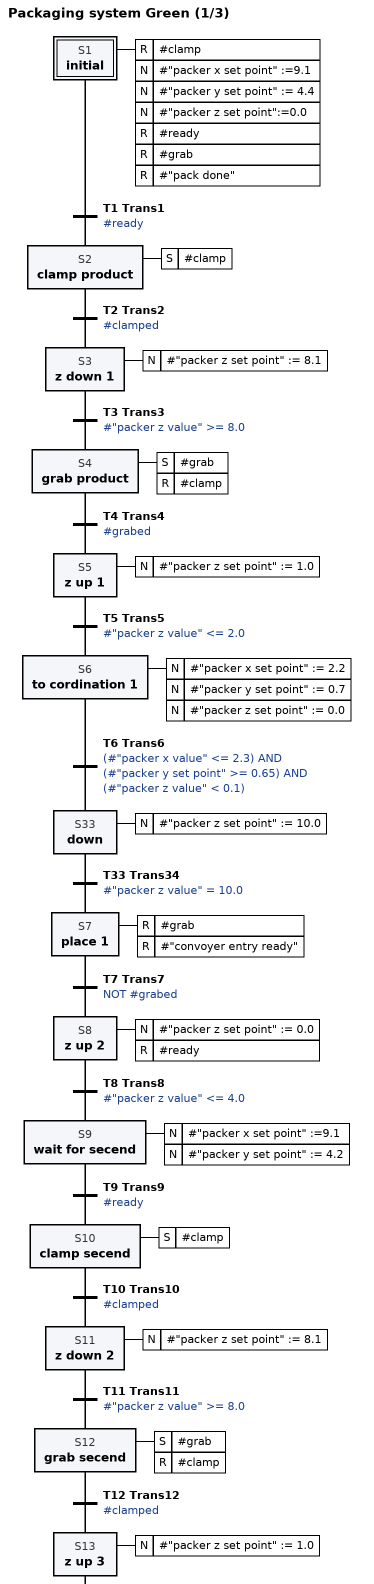
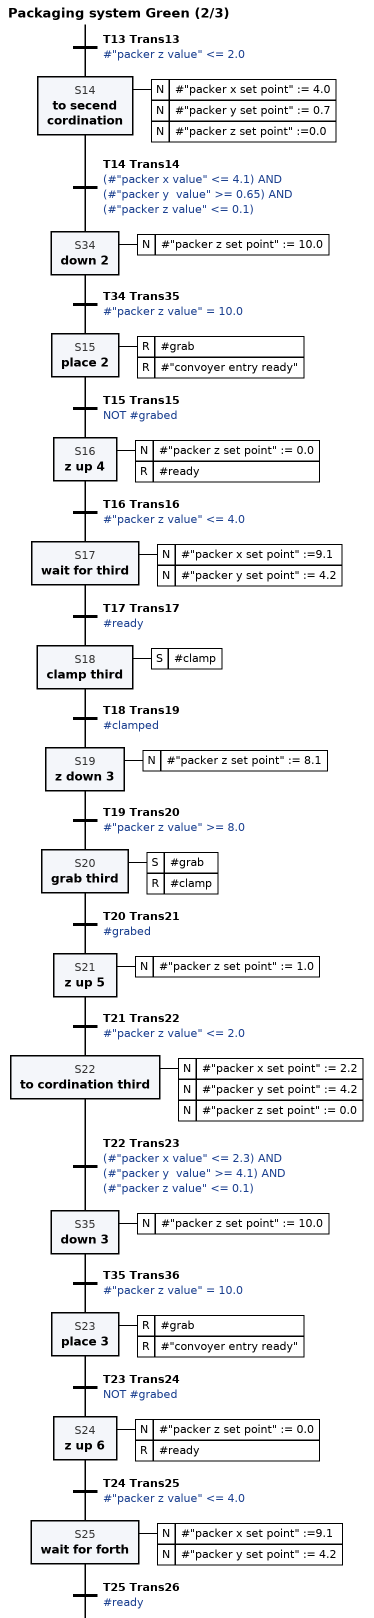
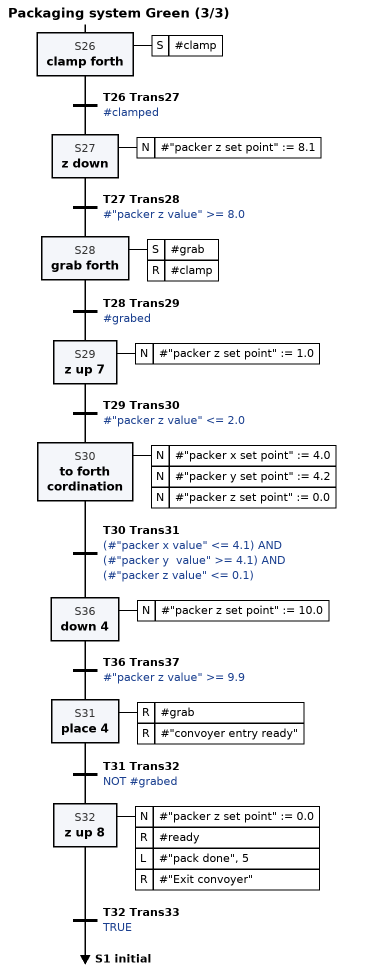
   // sequencer 1
   INITIAL_STEP initial:   // S1
              R    #clamp
              N    #"packer x set point" :=9.1
              N    #"packer y set point" := 4.4
              N    #"packer z set point":=0.0
              R    #ready
              R    #grab
              R    #"pack done"
   END_STEP
   TRANSITION Trans1 FROM initial TO "clamp product"   // T1
      := #ready;
   END_TRANSITION
   STEP "clamp product":   // S2
              S    #clamp
   END_STEP
   TRANSITION Trans2 FROM "clamp product" TO "z down 1"   // T2
      := #clamped;
   END_TRANSITION
   STEP "z down 1":   // S3
              N    #"packer z set point" := 8.1
   END_STEP
   TRANSITION Trans3 FROM "z down 1" TO "grab product"   // T3
      := #"packer z value" >= 8.0;
   END_TRANSITION
   STEP "grab product":   // S4
              S    #grab
              R    #clamp
   END_STEP
   TRANSITION Trans4 FROM "grab product" TO "z up 1"   // T4
      := #grabed;
   END_TRANSITION
   STEP "z up 1":   // S5
              N    #"packer z set point" := 1.0
   END_STEP
   TRANSITION Trans5 FROM "z up 1" TO "to cordination 1"   // T5
      := #"packer z value" <= 2.0;
   END_TRANSITION
   STEP "to cordination 1":   // S6
              N    #"packer x set point" := 2.2
              N    #"packer y set point" := 0.7
              N    #"packer z set point" := 0.0
   END_STEP
   TRANSITION Trans6 FROM "to cordination 1" TO down   // T6
      := (#"packer x value" <= 2.3) AND (#"packer y set point" >= 0.65) AND (#"packer z value" < 0.1);
   END_TRANSITION
   STEP "place 1":   // S7
              R    #grab
              R    #"convoyer entry ready"
   END_STEP
   TRANSITION Trans7 FROM "place 1" TO "z up 2"   // T7
      := NOT #grabed;
   END_TRANSITION
   STEP "z up 2":   // S8
              N    #"packer z set point" := 0.0
              R    #ready
   END_STEP
   TRANSITION Trans8 FROM "z up 2" TO "wait for secend"   // T8
      := #"packer z value" <= 4.0;
   END_TRANSITION
   STEP "wait for secend":   // S9
              N    #"packer x set point" :=9.1
              N    #"packer y set point" := 4.2
   END_STEP
   TRANSITION Trans9 FROM "wait for secend" TO "clamp secend"   // T9
      := #ready;
   END_TRANSITION
   STEP "clamp secend":   // S10
              S    #clamp
   END_STEP
   TRANSITION Trans10 FROM "clamp secend" TO "z down 2"   // T10
      := #clamped;
   END_TRANSITION
   STEP "z down 2":   // S11
              N    #"packer z set point" := 8.1
   END_STEP
   TRANSITION Trans11 FROM "z down 2" TO "grab secend"   // T11
      := #"packer z value" >= 8.0;
   END_TRANSITION
   STEP "grab secend":   // S12
              S    #grab
              R    #clamp
   END_STEP
   TRANSITION Trans12 FROM "grab secend" TO "z up 3"   // T12
      := #clamped;
   END_TRANSITION
   STEP "z up 3":   // S13
              N    #"packer z set point" := 1.0
   END_STEP
   TRANSITION Trans13 FROM "z up 3" TO "to secend cordination"   // T13
      := #"packer z value" <= 2.0;
   END_TRANSITION
   STEP "to secend cordination":   // S14
              N    #"packer x set point" := 4.0
              N    #"packer y set point" := 0.7
              N    #"packer z set point" :=0.0
   END_STEP
   TRANSITION Trans14 FROM "to secend cordination" TO "down 2"   // T14
      := (#"packer x value" <= 4.1) AND (#"packer y  value" >= 0.65) AND (#"packer z value" <= 0.1);
   END_TRANSITION
   STEP "place 2":   // S15
              R    #grab
              R    #"convoyer entry ready"
   END_STEP
   TRANSITION Trans15 FROM "place 2" TO "z up 4"   // T15
      := NOT #grabed;
   END_TRANSITION
   STEP "z up 4":   // S16
              N    #"packer z set point" := 0.0
              R    #ready
   END_STEP
   TRANSITION Trans16 FROM "z up 4" TO "wait for third"   // T16
      := #"packer z value" <= 4.0;
   END_TRANSITION
   STEP "wait for third":   // S17
              N    #"packer x set point" :=9.1
              N    #"packer y set point" := 4.2
   END_STEP
   TRANSITION Trans17 FROM "wait for third" TO "clamp third"   // T17
      := #ready;
   END_TRANSITION
   STEP "grab third":   // S20
              S    #grab
              R    #clamp
   END_STEP
   TRANSITION Trans21 FROM "grab third" TO "z up 5"   // T20
      := #grabed;
   END_TRANSITION
   STEP "clamp third":   // S18
              S    #clamp
   END_STEP
   TRANSITION Trans19 FROM "clamp third" TO "z down 3"   // T18
      := #clamped;
   END_TRANSITION
   STEP "z down 3":   // S19
              N    #"packer z set point" := 8.1
   END_STEP
   TRANSITION Trans20 FROM "z down 3" TO "grab third"   // T19
      := #"packer z value" >= 8.0;
   END_TRANSITION
   STEP "z up 5":   // S21
              N    #"packer z set point" := 1.0
   END_STEP
   TRANSITION Trans22 FROM "z up 5" TO "to cordination third"   // T21
      := #"packer z value" <= 2.0;
   END_TRANSITION
   STEP "to cordination third":   // S22
              N    #"packer x set point" := 2.2
              N    #"packer y set point" := 4.2
              N    #"packer z set point" := 0.0
   END_STEP
   TRANSITION Trans23 FROM "to cordination third" TO "down 3"   // T22
      := (#"packer x value" <= 2.3) AND (#"packer y  value" >= 4.1) AND (#"packer z value" <= 0.1);
   END_TRANSITION
   STEP "place 3":   // S23
              R    #grab
              R    #"convoyer entry ready"
   END_STEP
   TRANSITION Trans24 FROM "place 3" TO "z up 6"   // T23
      := NOT #grabed;
   END_TRANSITION
   STEP "z up 6":   // S24
              N    #"packer z set point" := 0.0
              R    #ready
   END_STEP
   TRANSITION Trans25 FROM "z up 6" TO "wait for forth"   // T24
      := #"packer z value" <= 4.0;
   END_TRANSITION
   STEP "wait for forth":   // S25
              N    #"packer x set point" :=9.1
              N    #"packer y set point" := 4.2
   END_STEP
   TRANSITION Trans26 FROM "wait for forth" TO "clamp forth"   // T25
      := #ready;
   END_TRANSITION
   STEP "clamp forth":   // S26
              S    #clamp
   END_STEP
   TRANSITION Trans27 FROM "clamp forth" TO "z down"   // T26
      := #clamped;
   END_TRANSITION
   STEP "z down":   // S27
              N    #"packer z set point" := 8.1
   END_STEP
   TRANSITION Trans28 FROM "z down" TO "grab forth"   // T27
      := #"packer z value" >= 8.0;
   END_TRANSITION
   STEP "grab forth":   // S28
              S    #grab
              R    #clamp
   END_STEP
   TRANSITION Trans29 FROM "grab forth" TO "z up 7"   // T28
      := #grabed;
   END_TRANSITION
   STEP "z up 7":   // S29
              N    #"packer z set point" := 1.0
   END_STEP
   TRANSITION Trans30 FROM "z up 7" TO "to forth cordination"   // T29
      := #"packer z value" <= 2.0;
   END_TRANSITION
   STEP "to forth cordination":   // S30
              N    #"packer x set point" := 4.0
              N    #"packer y set point" := 4.2
              N    #"packer z set point" := 0.0
   END_STEP
   TRANSITION Trans31 FROM "to forth cordination" TO "down 4"   // T30
      := (#"packer x value" <= 4.1) AND (#"packer y  value" >= 4.1) AND (#"packer z value" <= 0.1);
   END_TRANSITION
   STEP "place 4":   // S31
              R    #grab
              R    #"convoyer entry ready"
   END_STEP
   TRANSITION Trans32 FROM "place 4" TO "z up 8"   // T31
      := NOT #grabed;
   END_TRANSITION
   STEP "z up 8":   // S32
              N    #"packer z set point" := 0.0
              R    #ready
              L    #"pack done", 5
              R    #"Exit convoyer"
   END_STEP
   TRANSITION Trans33 FROM "z up 8" TO initial   // T32, jump
      := TRUE;
   END_TRANSITION
   STEP down:   // S33
              N    #"packer z set point" := 10.0
   END_STEP
   TRANSITION Trans34 FROM down TO "place 1"   // T33
      := #"packer z value" = 10.0;
   END_TRANSITION
   STEP "down 2":   // S34
              N    #"packer z set point" := 10.0
   END_STEP
   TRANSITION Trans35 FROM "down 2" TO "place 2"   // T34
      := #"packer z value" = 10.0;
   END_TRANSITION
   STEP "down 3":   // S35
              N    #"packer z set point" := 10.0
   END_STEP
   TRANSITION Trans36 FROM "down 3" TO "place 3"   // T35
      := #"packer z value" = 10.0;
   END_TRANSITION
   STEP "down 4":   // S36
              N    #"packer z set point" := 10.0
   END_STEP
   TRANSITION Trans37 FROM "down 4" TO "place 4"   // T36
      := #"packer z value" >= 9.9;
   END_TRANSITION
END_FUNCTION_BLOCK

FUNCTION "packaging entry convoyers" : Void   // FC7, LAD
{ S7_Optimized_Access := 'FALSE' }
VERSION : 0.1
   VAR_TEMP   // added for the SCL form of the ladder/FBD networks
      _w1 : Bool;
      _s5time1 : S5Time;
   END_VAR
BEGIN

REGION Network 1: Blue Assemble Exit Convoyer 1
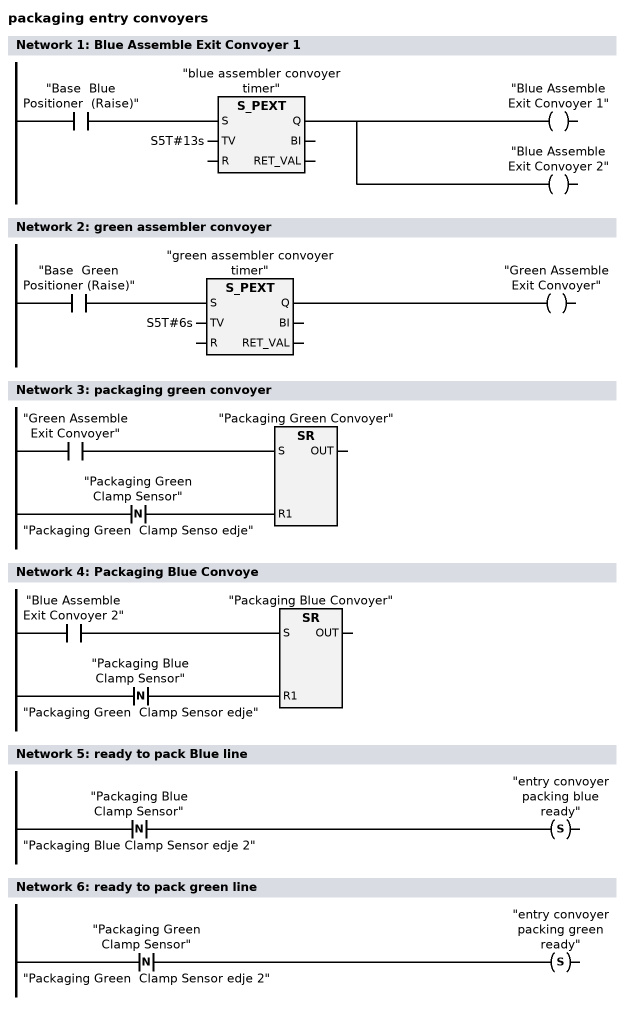
   RUNG wire#powerrail
      Contact( "Base  Blue Positioner  (Raise)" )
      S_PEXT(T_NO := "blue assembler convoyer timer", TV := S5T#13s, R :=, BI =>, RET_VAL =>)
      wire#w1
      Coil( "Blue Assemble Exit Convoyer 1" )
   END_RUNG
   RUNG wire#w1
      Coil( "Blue Assemble Exit Convoyer 2" )
   END_RUNG
   // the same network as SCL:
   #_s5time1 := S_PEXT(T_NO := "blue assembler convoyer timer",
                       S := "Base  Blue Positioner  (Raise)",
                       TV := S5T#13s,
                       Q => #_w1);
   "Blue Assemble Exit Convoyer 1" := #_w1;
   "Blue Assemble Exit Convoyer 2" := #_w1;
END_REGION

REGION Network 2: green assembler convoyer
   RUNG wire#powerrail
      Contact( "Base  Green Positioner (Raise)" )
      S_PEXT(T_NO := "green assembler convoyer timer", TV := S5T#6s, R :=, BI =>, RET_VAL =>)
      Coil( "Green Assemble Exit Convoyer" )
   END_RUNG
   // the same network as SCL:
   #_s5time1 := S_PEXT(T_NO := "green assembler convoyer timer",
                       S := "Base  Green Positioner (Raise)",
                       TV := S5T#6s,
                       Q => #_w1);
   "Green Assemble Exit Convoyer" := #_w1;
END_REGION

REGION Network 3: packaging green convoyer
   RUNG wire#powerrail
      Contact( "Green Assemble Exit Convoyer" )
      S_SR(operand := "Packaging Green Convoyer", r1 := wire#w1)
   END_RUNG
   RUNG wire#powerrail
      N_Contact(operand := "Packaging Green  Clamp Sensor", bit := "Packaging Green  Clamp Senso edje")
   END_RUNG wire#w1
   // the same network as SCL:
   #_w1 := NOT "Packaging Green  Clamp Sensor" AND "Packaging Green  Clamp Senso edje";   // falling edge of "Packaging Green  Clamp Sensor"
   "Packaging Green  Clamp Senso edje" := "Packaging Green  Clamp Sensor";
   IF "Green Assemble Exit Convoyer" THEN
       "Packaging Green Convoyer" := TRUE;   // SR flip-flop
   END_IF;
   IF #_w1 THEN "Packaging Green Convoyer" := FALSE; END_IF;
END_REGION

REGION Network 4: Packaging Blue Convoye
   RUNG wire#powerrail
      Contact( "Blue Assemble Exit Convoyer 2" )
      S_SR(operand := "Packaging Blue Convoyer", r1 := wire#w1)
   END_RUNG
   RUNG wire#powerrail
      N_Contact(operand := "Packaging Blue Clamp Sensor", bit := "Packaging Green  Clamp Sensor edje")
   END_RUNG wire#w1
   // the same network as SCL:
   #_w1 := NOT "Packaging Blue Clamp Sensor" AND "Packaging Green  Clamp Sensor edje";   // falling edge of "Packaging Blue Clamp Sensor"
   "Packaging Green  Clamp Sensor edje" := "Packaging Blue Clamp Sensor";
   IF "Blue Assemble Exit Convoyer 2" THEN
       "Packaging Blue Convoyer" := TRUE;   // SR flip-flop
   END_IF;
   IF #_w1 THEN "Packaging Blue Convoyer" := FALSE; END_IF;
END_REGION

REGION Network 5: ready to pack Blue line
   RUNG wire#powerrail
      N_Contact(operand := "Packaging Blue Clamp Sensor", bit := "Packaging Blue Clamp Sensor edje 2")
      S_Coil( "entry convoyer packing blue ready" )
   END_RUNG
   // the same network as SCL:
   #_w1 := NOT "Packaging Blue Clamp Sensor" AND "Packaging Blue Clamp Sensor edje 2";   // falling edge of "Packaging Blue Clamp Sensor"
   "Packaging Blue Clamp Sensor edje 2" := "Packaging Blue Clamp Sensor";
   IF #_w1 THEN "entry convoyer packing blue ready" := TRUE; END_IF;
END_REGION

REGION Network 6: ready to pack green line
   RUNG wire#powerrail
      N_Contact(operand := "Packaging Green  Clamp Sensor", bit := "Packaging Green  Clamp Sensor edje 2")
      S_Coil( "entry convoyer packing green ready" )
   END_RUNG
   // the same network as SCL:
   #_w1 := NOT "Packaging Green  Clamp Sensor" AND "Packaging Green  Clamp Sensor edje 2";   // falling edge of "Packaging Green  Clamp Sensor"
   "Packaging Green  Clamp Sensor edje 2" := "Packaging Green  Clamp Sensor";
   IF #_w1 THEN "entry convoyer packing green ready" := TRUE; END_IF;
END_REGION
END_FUNCTION

FUNCTION "Packaging" : Void   // FC8, LAD
{ S7_Optimized_Access := 'FALSE' }
VERSION : 0.1
BEGIN

REGION Network 1: Packing entry convoyers
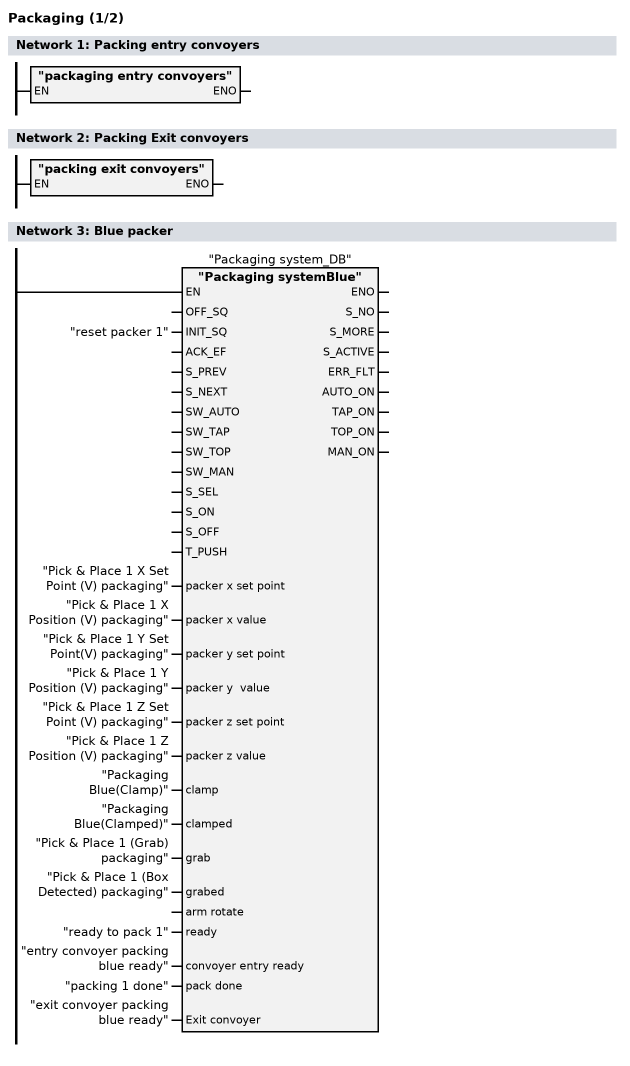
   RUNG wire#powerrail
      "packaging entry convoyers"()
   END_RUNG
   // the same network as SCL:
   "packaging entry convoyers"();
END_REGION

REGION Network 2: Packing Exit convoyers
   RUNG wire#powerrail
      "packing exit convoyers"()
   END_RUNG
   // the same network as SCL:
   "packing exit convoyers"();
END_REGION

REGION Network 3: Blue packer
   RUNG wire#powerrail
      "Packaging system_DB"(OFF_SQ :=, INIT_SQ := "reset packer 1", ACK_EF :=, S_PREV :=, S_NEXT :=, SW_AUTO :=, SW_TAP :=, SW_TOP :=, SW_MAN :=, S_SEL :=, S_ON :=, S_OFF :=, T_PUSH :=, "packer x set point" := "Pick & Place 1 X Set Point (V) packaging", "packer x value" := "Pick & Place 1 X Position (V) packaging", "packer y set point" := "Pick & Place 1 Y Set Point(V) packaging", "packer y  value" := "Pick & Place 1 Y Position (V) packaging", "packer z set point" := "Pick & Place 1 Z Set Point (V) packaging", "packer z value" := "Pick & Place 1 Z Position (V) packaging", clamp := "Packaging Blue(Clamp)", clamped := "Packaging Blue(Clamped)", grab := "Pick & Place 1 (Grab) packaging", grabed := "Pick & Place 1 (Box Detected) packaging", "arm rotate" :=, ready := "ready to pack 1", "convoyer entry ready" := "entry convoyer packing blue ready", "pack done" := "packing 1 done", "Exit convoyer" := "exit convoyer packing blue ready", S_NO =>, S_MORE =>, S_ACTIVE =>, ERR_FLT =>, AUTO_ON =>, TAP_ON =>, TOP_ON =>, MAN_ON =>)
   END_RUNG
   // the same network as SCL:
   "Packaging system_DB"(INIT_SQ := "reset packer 1",   // "Packaging systemBlue"
                         "packer x set point" := "Pick & Place 1 X Set Point (V) packaging",
                         "packer x value" := "Pick & Place 1 X Position (V) packaging",
                         "packer y set point" := "Pick & Place 1 Y Set Point(V) packaging",
                         "packer y  value" := "Pick & Place 1 Y Position (V) packaging",
                         "packer z set point" := "Pick & Place 1 Z Set Point (V) packaging",
                         "packer z value" := "Pick & Place 1 Z Position (V) packaging",
                         clamp := "Packaging Blue(Clamp)",
                         clamped := "Packaging Blue(Clamped)",
                         grab := "Pick & Place 1 (Grab) packaging",
                         grabed := "Pick & Place 1 (Box Detected) packaging",
                         ready := "ready to pack 1",
                         "convoyer entry ready" := "entry convoyer packing blue ready",
                         "pack done" := "packing 1 done",
                         "Exit convoyer" := "exit convoyer packing blue ready");
END_REGION

REGION Network 4: Green packer
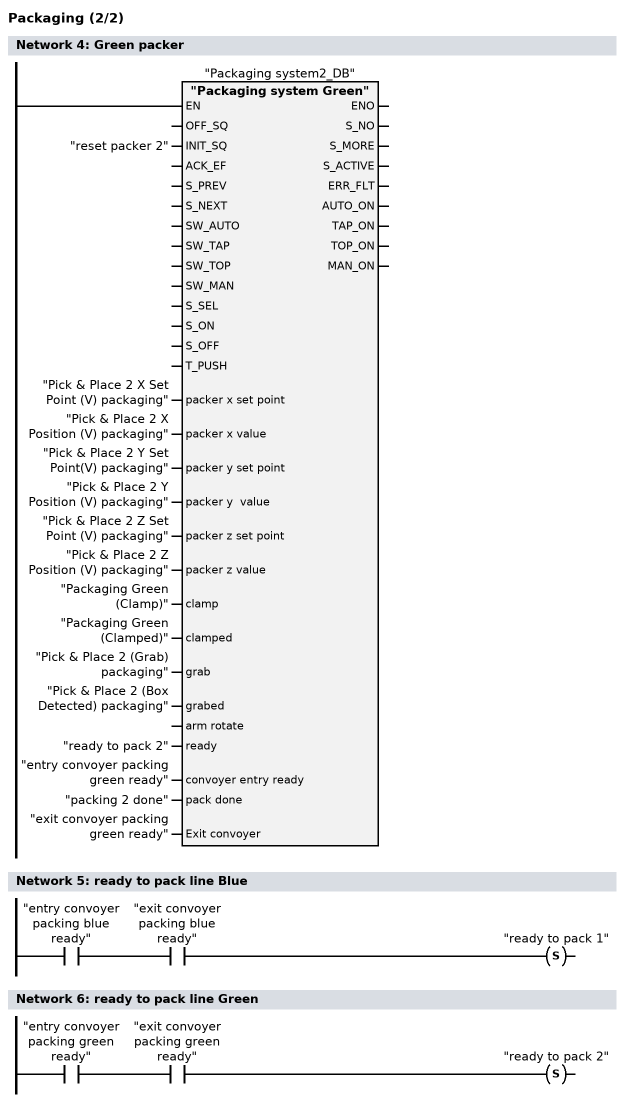
   RUNG wire#powerrail
      "Packaging system2_DB"(OFF_SQ :=, INIT_SQ := "reset packer 2", ACK_EF :=, S_PREV :=, S_NEXT :=, SW_AUTO :=, SW_TAP :=, SW_TOP :=, SW_MAN :=, S_SEL :=, S_ON :=, S_OFF :=, T_PUSH :=, "packer x set point" := "Pick & Place 2 X Set Point (V) packaging", "packer x value" := "Pick & Place 2 X Position (V) packaging", "packer y set point" := "Pick & Place 2 Y Set Point(V) packaging", "packer y  value" := "Pick & Place 2 Y Position (V) packaging", "packer z set point" := "Pick & Place 2 Z Set Point (V) packaging", "packer z value" := "Pick & Place 2 Z Position (V) packaging", clamp := "Packaging Green (Clamp)", clamped := "Packaging Green (Clamped)", grab := "Pick & Place 2 (Grab) packaging", grabed := "Pick & Place 2 (Box Detected) packaging", "arm rotate" :=, ready := "ready to pack 2", "convoyer entry ready" := "entry convoyer packing green ready", "pack done" := "packing 2 done", "Exit convoyer" := "exit convoyer packing green ready", S_NO =>, S_MORE =>, S_ACTIVE =>, ERR_FLT =>, AUTO_ON =>, TAP_ON =>, TOP_ON =>, MAN_ON =>)
   END_RUNG
   // the same network as SCL:
   "Packaging system2_DB"(INIT_SQ := "reset packer 2",   // "Packaging system Green"
                          "packer x set point" := "Pick & Place 2 X Set Point (V) packaging",
                          "packer x value" := "Pick & Place 2 X Position (V) packaging",
                          "packer y set point" := "Pick & Place 2 Y Set Point(V) packaging",
                          "packer y  value" := "Pick & Place 2 Y Position (V) packaging",
                          "packer z set point" := "Pick & Place 2 Z Set Point (V) packaging",
                          "packer z value" := "Pick & Place 2 Z Position (V) packaging",
                          clamp := "Packaging Green (Clamp)",
                          clamped := "Packaging Green (Clamped)",
                          grab := "Pick & Place 2 (Grab) packaging",
                          grabed := "Pick & Place 2 (Box Detected) packaging",
                          ready := "ready to pack 2",
                          "convoyer entry ready" := "entry convoyer packing green ready",
                          "pack done" := "packing 2 done",
                          "Exit convoyer" := "exit convoyer packing green ready");
END_REGION

REGION Network 5: ready to pack line Blue
   RUNG wire#powerrail
      Contact( "entry convoyer packing blue ready" )
      Contact( "exit convoyer packing blue ready" )
      S_Coil( "ready to pack 1" )
   END_RUNG
   // the same network as SCL:
   IF "entry convoyer packing blue ready" AND "exit convoyer packing blue ready" THEN
       "ready to pack 1" := TRUE;
   END_IF;
END_REGION

REGION Network 6: ready to pack line Green
   RUNG wire#powerrail
      Contact( "entry convoyer packing green ready" )
      Contact( "exit convoyer packing green ready" )
      S_Coil( "ready to pack 2" )
   END_RUNG
   // the same network as SCL:
   IF "entry convoyer packing green ready" AND "exit convoyer packing green ready" THEN
       "ready to pack 2" := TRUE;
   END_IF;
END_REGION
END_FUNCTION

FUNCTION "packing exit convoyers" : Void   // FC9, LAD
{ S7_Optimized_Access := 'FALSE' }
VERSION : 0.1
   VAR_TEMP   // added for the SCL form of the ladder/FBD networks
      _w1 : Bool;
   END_VAR
BEGIN

REGION Network 1: exit convoyer 1 Blue
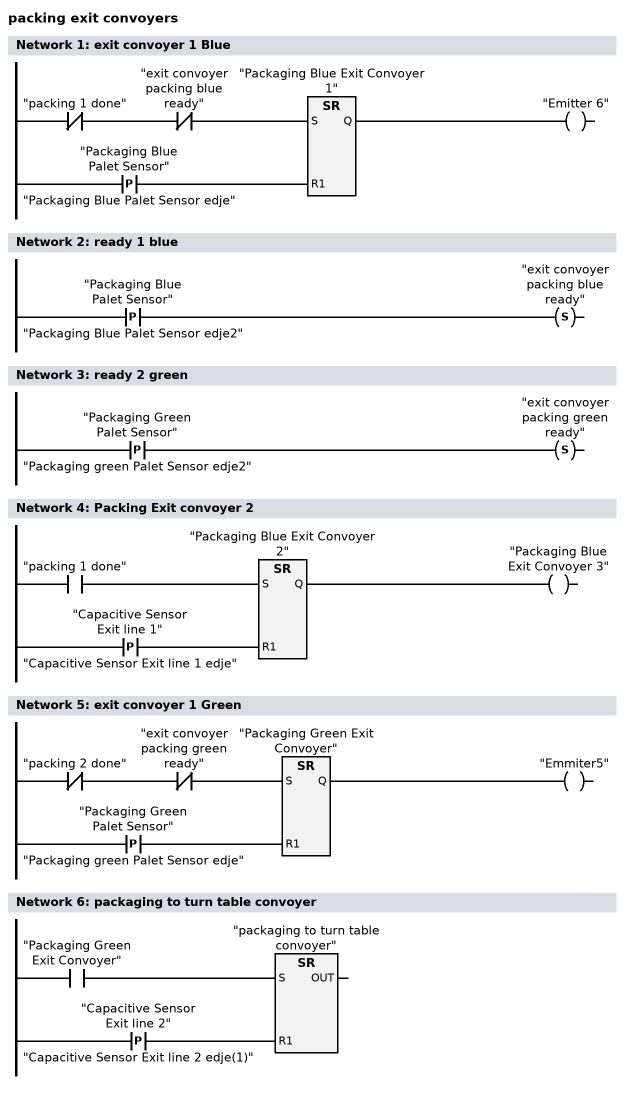
   RUNG wire#powerrail
      I_Contact( "packing 1 done" )
      I_Contact( "exit convoyer packing blue ready" )
      S_SR(operand := "Packaging Blue Exit Convoyer 1", r1 := wire#w1)
      Coil( "Emitter 6" )
   END_RUNG
   RUNG wire#powerrail
      P_Contact(operand := "Packaging Blue Palet Sensor", bit := "Packaging Blue Palet Sensor edje")
   END_RUNG wire#w1
   // the same network as SCL:
   #_w1 := "Packaging Blue Palet Sensor" AND NOT "Packaging Blue Palet Sensor edje";   // rising edge of "Packaging Blue Palet Sensor"
   "Packaging Blue Palet Sensor edje" := "Packaging Blue Palet Sensor";
   IF NOT "packing 1 done" AND NOT "exit convoyer packing blue ready" THEN
       "Packaging Blue Exit Convoyer 1" := TRUE;   // SR flip-flop
   END_IF;
   IF #_w1 THEN "Packaging Blue Exit Convoyer 1" := FALSE; END_IF;
   "Emitter 6" := "Packaging Blue Exit Convoyer 1";
END_REGION

REGION Network 2: ready 1 blue
   RUNG wire#powerrail
      P_Contact(operand := "Packaging Blue Palet Sensor", bit := "Packaging Blue Palet Sensor edje2")
      S_Coil( "exit convoyer packing blue ready" )
   END_RUNG
   // the same network as SCL:
   #_w1 := "Packaging Blue Palet Sensor" AND NOT "Packaging Blue Palet Sensor edje2";   // rising edge of "Packaging Blue Palet Sensor"
   "Packaging Blue Palet Sensor edje2" := "Packaging Blue Palet Sensor";
   IF #_w1 THEN "exit convoyer packing blue ready" := TRUE; END_IF;
END_REGION

REGION Network 3: ready 2 green
   RUNG wire#powerrail
      P_Contact(operand := "Packaging Green  Palet Sensor", bit := "Packaging green Palet Sensor edje2")
      S_Coil( "exit convoyer packing green ready" )
   END_RUNG
   // the same network as SCL:
   #_w1 := "Packaging Green  Palet Sensor" AND NOT "Packaging green Palet Sensor edje2";   // rising edge of "Packaging Green  Palet Sensor"
   "Packaging green Palet Sensor edje2" := "Packaging Green  Palet Sensor";
   IF #_w1 THEN "exit convoyer packing green ready" := TRUE; END_IF;
END_REGION

REGION Network 4: Packing Exit convoyer 2
   RUNG wire#powerrail
      Contact( "packing 1 done" )
      S_SR(operand := "Packaging Blue Exit Convoyer 2", r1 := wire#w1)
      Coil( "Packaging Blue Exit Convoyer 3" )
   END_RUNG
   RUNG wire#powerrail
      P_Contact(operand := "Capacitive Sensor Exit line 1", bit := "Capacitive Sensor Exit line 1 edje")
   END_RUNG wire#w1
   // the same network as SCL:
   #_w1 := "Capacitive Sensor Exit line 1" AND NOT "Capacitive Sensor Exit line 1 edje";   // rising edge of "Capacitive Sensor Exit line 1"
   "Capacitive Sensor Exit line 1 edje" := "Capacitive Sensor Exit line 1";
   IF "packing 1 done" THEN
       "Packaging Blue Exit Convoyer 2" := TRUE;   // SR flip-flop
   END_IF;
   IF #_w1 THEN "Packaging Blue Exit Convoyer 2" := FALSE; END_IF;
   "Packaging Blue Exit Convoyer 3" := "Packaging Blue Exit Convoyer 2";
END_REGION

REGION Network 5: exit convoyer 1 Green
   RUNG wire#powerrail
      I_Contact( "packing 2 done" )
      I_Contact( "exit convoyer packing green ready" )
      S_SR(operand := "Packaging Green Exit Convoyer", r1 := wire#w1)
      Coil( "Emmiter5" )
   END_RUNG
   RUNG wire#powerrail
      P_Contact(operand := "Packaging Green  Palet Sensor", bit := "Packaging green Palet Sensor edje")
   END_RUNG wire#w1
   // the same network as SCL:
   #_w1 := "Packaging Green  Palet Sensor" AND NOT "Packaging green Palet Sensor edje";   // rising edge of "Packaging Green  Palet Sensor"
   "Packaging green Palet Sensor edje" := "Packaging Green  Palet Sensor";
   IF NOT "packing 2 done" AND NOT "exit convoyer packing green ready" THEN
       "Packaging Green Exit Convoyer" := TRUE;   // SR flip-flop
   END_IF;
   IF #_w1 THEN "Packaging Green Exit Convoyer" := FALSE; END_IF;
   "Emmiter5" := "Packaging Green Exit Convoyer";
END_REGION

REGION Network 6: packaging to turn table convoyer
   RUNG wire#powerrail
      Contact( "Packaging Green Exit Convoyer" )
      S_SR(operand := "packaging to turn table convoyer", r1 := wire#w1)
   END_RUNG
   RUNG wire#powerrail
      P_Contact(operand := "Capacitive Sensor Exit line 2", bit := "Capacitive Sensor Exit line 2 edje(1)")
   END_RUNG wire#w1
   // the same network as SCL:
   #_w1 := "Capacitive Sensor Exit line 2" AND NOT "Capacitive Sensor Exit line 2 edje(1)";   // rising edge of "Capacitive Sensor Exit line 2"
   "Capacitive Sensor Exit line 2 edje(1)" := "Capacitive Sensor Exit line 2";
   IF "Packaging Green Exit Convoyer" THEN
       "packaging to turn table convoyer" := TRUE;   // SR flip-flop
   END_IF;
   IF #_w1 THEN "packaging to turn table convoyer" := FALSE; END_IF;
END_REGION
END_FUNCTION

// folder: Sort And Assemble

